  [1014] = {x=-21.274, y=-6.415, z=129.21, rx=179.838, ry=0.326, rz=-127.185, fatherId=FrmDraw[0]}
  [1015] = {x=-21.178, y=-6.199, z=129.218, rx=179.848, ry=0.308, rz=-127.673, fatherId=FrmDraw[0]}
  [1016] = {x=-21.058, y=-5.968, z=129.228, rx=179.861, ry=0.287, rz=-128.317, fatherId=FrmDraw[0]}
  [1017] = {x=-20.945, y=-5.787, z=129.236, rx=179.872, ry=0.268, rz=-128.961, fatherId=FrmDraw[0]}
  [1018] = {x=-20.8, y=-5.61, z=129.247, rx=179.886, ry=0.243, rz=-129.828, fatherId=FrmDraw[0]}
  [1019] = {x=-20.652, y=-5.478, z=129.258, rx=179.9, ry=0.219, rz=-130.741, fatherId=FrmDraw[0]}
  [1020] = {x=-20.476, y=-5.365, z=129.27, rx=179.915, ry=0.19, rz=-131.877, fatherId=FrmDraw[0]}
  [1021] = {x=-20.289, y=-5.287, z=129.282, rx=179.931, ry=0.16, rz=-133.12, fatherId=FrmDraw[0]}
  [1022] = {x=-20.088, y=-5.227, z=129.295, rx=179.946, ry=0.129, rz=-134.508, fatherId=FrmDraw[0]}
  [1023] = {x=-19.895, y=-5.156, z=129.306, rx=179.959, ry=0.102, rz=-135.941, fatherId=FrmDraw[0]}
  [1024] = {x=-19.715, y=-5.077, z=129.317, rx=179.969, ry=0.08, rz=-137.368, fatherId=FrmDraw[0]}
  [1025] = {x=-19.561, y=-4.999, z=129.326, rx=179.976, ry=0.063, rz=-138.682, fatherId=FrmDraw[0]}
  [1026] = {x=-19.427, y=-4.922, z=129.333, rx=179.982, ry=0.05, rz=-139.885, fatherId=FrmDraw[0]}
  [1027] = {x=-19.274, y=-4.826, z=129.341, rx=179.987, ry=0.038, rz=-141.341, fatherId=FrmDraw[0]}
  [1028] = {x=-19.151, y=-4.74, z=129.347, rx=179.99, ry=0.03, rz=-142.591, fatherId=FrmDraw[0]}
  [1029] = {x=-19.043, y=-4.661, z=129.352, rx=179.992, ry=0.024, rz=-143.734, fatherId=FrmDraw[0]}
  [1030] = {x=-18.902, y=-4.55, z=129.359, rx=179.994, ry=0.018, rz=-145.305, fatherId=FrmDraw[0]}
  [1031] = {x=-18.775, y=-4.444, z=129.365, rx=179.996, ry=0.014, rz=-146.807, fatherId=FrmDraw[0]}
  [1032] = {x=-18.658, y=-4.341, z=129.37, rx=179.997, ry=0.011, rz=-148.246, fatherId=FrmDraw[0]}
  [1033] = {x=-18.553, y=-4.238, z=129.374, rx=179.997, ry=0.01, rz=-149.624, fatherId=FrmDraw[0]}
  [1034] = {x=-18.457, y=-4.137, z=129.378, rx=179.997, ry=0.011, rz=-150.951, fatherId=FrmDraw[0]}
  [1035] = {x=-18.37, y=-4.037, z=129.381, rx=179.997, ry=0.012, rz=-152.231, fatherId=FrmDraw[0]}
  [1036] = {x=-18.29, y=-3.938, z=129.384, rx=179.996, ry=0.015, rz=-153.473, fatherId=FrmDraw[0]}
  [1037] = {x=-18.217, y=-3.841, z=129.387, rx=179.996, ry=0.02, rz=-154.679, fatherId=FrmDraw[0]}
  [1038] = {x=-18.151, y=-3.745, z=129.389, rx=179.995, ry=0.025, rz=-155.853, fatherId=FrmDraw[0]}
  [1039] = {x=-18.09, y=-3.651, z=129.39, rx=179.994, ry=0.031, rz=-157, fatherId=FrmDraw[0]}
  [1040] = {x=-18.035, y=-3.558, z=129.392, rx=179.993, ry=0.038, rz=-158.121, fatherId=FrmDraw[0]}
  [1041] = {x=-17.962, y=-3.424, z=129.393, rx=179.991, ry=0.049, rz=-159.732, fatherId=FrmDraw[0]}
  [1042] = {x=-17.898, y=-3.289, z=129.394, rx=179.99, ry=0.063, rz=-161.357, fatherId=FrmDraw[0]}
  [1043] = {x=-17.843, y=-3.162, z=129.394, rx=179.988, ry=0.078, rz=-162.916, fatherId=FrmDraw[0]}
  [1044] = {x=-17.795, y=-3.04, z=129.394, rx=179.987, ry=0.094, rz=-164.461, fatherId=FrmDraw[0]}
  [1045] = {x=-17.752, y=-2.925, z=129.393, rx=179.986, ry=0.111, rz=-165.983, fatherId=FrmDraw[0]}
  [1046] = {x=-17.715, y=-2.816, z=129.392, rx=179.986, ry=0.128, rz=-167.488, fatherId=FrmDraw[0]}
  [1047] = {x=-17.683, y=-2.713, z=129.391, rx=179.986, ry=0.146, rz=-168.981, fatherId=FrmDraw[0]}
  [1048] = {x=-17.654, y=-2.616, z=129.389, rx=179.986, ry=0.164, rz=-170.464, fatherId=FrmDraw[0]}
  [1049] = {x=-17.63, y=-2.525, z=129.388, rx=179.987, ry=0.183, rz=-171.939, fatherId=FrmDraw[0]}
  [1050] = {x=-17.608, y=-2.44, z=129.386, rx=179.988, ry=0.202, rz=-173.407, fatherId=FrmDraw[0]}
  [1051] = {x=-17.59, y=-2.36, z=129.383, rx=179.99, ry=0.221, rz=-174.871, fatherId=FrmDraw[0]}
  [1052] = {x=-17.574, y=-2.286, z=129.381, rx=179.992, ry=0.241, rz=-176.331, fatherId=FrmDraw[0]}
  [1053] = {x=-17.563, y=-2.215, z=129.378, rx=179.995, ry=0.261, rz=-177.777, fatherId=FrmDraw[0]}
  [1054] = {x=-17.557, y=-2.118, z=129.374, rx=179.999, ry=0.29, rz=-179.658, fatherId=FrmDraw[0]}
  [1055] = {x=-17.561, y=-2.02, z=129.368, rx=-179.996, ry=0.321, rz=178.508, fatherId=FrmDraw[0]}
  [1056] = {x=-17.575, y=-1.922, z=129.363, rx=-179.99, ry=0.354, rz=176.715, fatherId=FrmDraw[0]}
  [1057] = {x=-17.597, y=-1.824, z=129.356, rx=-179.983, ry=0.389, rz=174.957, fatherId=FrmDraw[0]}
  [1058] = {x=-17.628, y=-1.725, z=129.349, rx=-179.975, ry=0.426, rz=173.239, fatherId=FrmDraw[0]}
  [1059] = {x=-17.665, y=-1.624, z=129.342, rx=-179.966, ry=0.463, rz=171.562, fatherId=FrmDraw[0]}
  [1060] = {x=-17.705, y=-1.521, z=129.334, rx=-179.956, ry=0.5, rz=169.92, fatherId=FrmDraw[0]}
  [1061] = {x=-17.745, y=-1.417, z=129.327, rx=-179.945, ry=0.534, rz=168.309, fatherId=FrmDraw[0]}
  [1062] = {x=-17.784, y=-1.312, z=129.32, rx=-179.934, ry=0.566, rz=166.727, fatherId=FrmDraw[0]}
  [1063] = {x=-17.822, y=-1.201, z=129.313, rx=-179.923, ry=0.596, rz=165.189, fatherId=FrmDraw[0]}
  [1064] = {x=-17.86, y=-1.084, z=129.307, rx=-179.911, ry=0.624, rz=163.696, fatherId=FrmDraw[0]}
  [1065] = {x=-17.899, y=-0.961, z=129.301, rx=-179.898, ry=0.651, rz=162.246, fatherId=FrmDraw[0]}
  [1066] = {x=-17.941, y=-0.832, z=129.295, rx=-179.886, ry=0.676, rz=160.836, fatherId=FrmDraw[0]}
  [1067] = {x=-17.986, y=-0.698, z=129.289, rx=-179.873, ry=0.702, rz=159.465, fatherId=FrmDraw[0]}
  [1068] = {x=-18.036, y=-0.559, z=129.283, rx=-179.86, ry=0.727, rz=158.13, fatherId=FrmDraw[0]}
  [1069] = {x=-18.09, y=-0.416, z=129.276, rx=-179.846, ry=0.752, rz=156.83, fatherId=FrmDraw[0]}
  [1070] = {x=-18.15, y=-0.268, z=129.269, rx=-179.831, ry=0.779, rz=155.562, fatherId=FrmDraw[0]}
  [1071] = {x=-18.216, y=-0.116, z=129.262, rx=-179.816, ry=0.806, rz=154.324, fatherId=FrmDraw[0]}
  [1072] = {x=-18.289, y=0.038, z=129.255, rx=-179.8, ry=0.835, rz=153.111, fatherId=FrmDraw[0]}
  [1073] = {x=-18.367, y=0.189, z=129.247, rx=-179.784, ry=0.864, rz=151.895, fatherId=FrmDraw[0]}
  [1074] = {x=-18.45, y=0.336, z=129.239, rx=-179.766, ry=0.893, rz=150.671, fatherId=FrmDraw[0]}
  [1075] = {x=-18.536, y=0.479, z=129.231, rx=-179.748, ry=0.922, rz=149.437, fatherId=FrmDraw[0]}
  [1076] = {x=-18.626, y=0.618, z=129.223, rx=-179.729, ry=0.951, rz=148.192, fatherId=FrmDraw[0]}
  [1077] = {x=-18.72, y=0.753, z=129.215, rx=-179.709, ry=0.98, rz=146.934, fatherId=FrmDraw[0]}
  [1078] = {x=-18.817, y=0.883, z=129.206, rx=-179.688, ry=1.008, rz=145.662, fatherId=FrmDraw[0]}
  [1079] = {x=-18.916, y=1.008, z=129.198, rx=-179.667, ry=1.036, rz=144.375, fatherId=FrmDraw[0]}
  [1080] = {x=-19.018, y=1.129, z=129.19, rx=-179.645, ry=1.062, rz=143.071, fatherId=FrmDraw[0]}
  [1081] = {x=-19.123, y=1.245, z=129.182, rx=-179.623, ry=1.088, rz=141.749, fatherId=FrmDraw[0]}
  [1082] = {x=-19.23, y=1.357, z=129.174, rx=-179.599, ry=1.113, rz=140.412, fatherId=FrmDraw[0]}
  [1083] = {x=-19.341, y=1.476, z=129.165, rx=-179.575, ry=1.139, rz=139.111, fatherId=FrmDraw[0]}
  [1084] = {x=-19.398, y=1.539, z=129.161, rx=-179.563, ry=1.152, rz=138.478, fatherId=FrmDraw[0]}
  [1085] = {x=-19.486, y=1.638, z=129.154, rx=-179.545, ry=1.172, rz=137.552, fatherId=FrmDraw[0]}
  [1086] = {x=-19.606, y=1.778, z=129.145, rx=-179.519, ry=1.2, rz=136.36, fatherId=FrmDraw[0]}
  [1087] = {x=-19.729, y=1.929, z=129.136, rx=-179.494, ry=1.229, rz=135.217, fatherId=FrmDraw[0]}
  [1088] = {x=-19.855, y=2.09, z=129.127, rx=-179.468, ry=1.258, rz=134.123, fatherId=FrmDraw[0]}
  [1089] = {x=-19.983, y=2.263, z=129.118, rx=-179.441, ry=1.287, rz=133.079, fatherId=FrmDraw[0]}
  [1090] = {x=-20.112, y=2.448, z=129.108, rx=-179.415, ry=1.316, rz=132.083, fatherId=FrmDraw[0]}
  [1091] = {x=-20.242, y=2.645, z=129.099, rx=-179.389, ry=1.345, rz=131.137, fatherId=FrmDraw[0]}
  [1092] = {x=-20.371, y=2.854, z=129.09, rx=-179.363, ry=1.374, rz=130.24, fatherId=FrmDraw[0]}
  [1093] = {x=-20.499, y=3.072, z=129.082, rx=-179.337, ry=1.401, rz=129.37, fatherId=FrmDraw[0]}
  [1094] = {x=-20.626, y=3.293, z=129.074, rx=-179.313, ry=1.425, rz=128.499, fatherId=FrmDraw[0]}
  [1095] = {x=-20.752, y=3.517, z=129.067, rx=-179.288, ry=1.448, rz=127.626, fatherId=FrmDraw[0]}
  [1096] = {x=-20.879, y=3.742, z=129.06, rx=-179.264, ry=1.468, rz=126.751, fatherId=FrmDraw[0]}
  [1097] = {x=-21.007, y=3.97, z=129.053, rx=-179.24, ry=1.487, rz=125.875, fatherId=FrmDraw[0]}
  [1098] = {x=-21.136, y=4.2, z=129.047, rx=-179.216, ry=1.505, rz=124.995, fatherId=FrmDraw[0]}
  [1099] = {x=-21.268, y=4.431, z=129.041, rx=-179.193, ry=1.522, rz=124.113, fatherId=FrmDraw[0]}
  [1100] = {x=-21.403, y=4.663, z=129.035, rx=-179.169, ry=1.538, rz=123.227, fatherId=FrmDraw[0]}
  [1101] = {x=-21.507, y=4.838, z=129.031, rx=-179.151, ry=1.55, rz=122.561, fatherId=FrmDraw[0]}
  [1102] = {x=-21.643, y=5.061, z=129.025, rx=-179.127, ry=1.566, rz=121.72, fatherId=FrmDraw[0]}
  [1103] = {x=-21.788, y=5.308, z=129.019, rx=-179.102, ry=1.583, rz=120.881, fatherId=FrmDraw[0]}
  [1104] = {x=-21.934, y=5.568, z=129.013, rx=-179.076, ry=1.603, rz=120.103, fatherId=FrmDraw[0]}
  [1105] = {x=-22.076, y=5.838, z=129.007, rx=-179.051, ry=1.623, rz=119.399, fatherId=FrmDraw[0]}
  [1106] = {x=-22.196, y=6.082, z=129.002, rx=-179.03, ry=1.642, rz=118.842, fatherId=FrmDraw[0]}
  [1107] = {x=-22.294, y=6.295, z=128.998, rx=-179.012, ry=1.657, rz=118.41, fatherId=FrmDraw[0]}
  [1108] = {x=-22.427, y=6.609, z=128.993, rx=-178.988, ry=1.679, rz=117.857, fatherId=FrmDraw[0]}
  [1109] = {x=-22.536, y=6.893, z=128.989, rx=-178.968, ry=1.698, rz=117.431, fatherId=FrmDraw[0]}
  [1110] = {x=-22.629, y=7.161, z=128.985, rx=-178.951, ry=1.714, rz=117.087, fatherId=FrmDraw[0]}
  [1111] = {x=-22.717, y=7.442, z=128.983, rx=-178.935, ry=1.73, rz=116.78, fatherId=FrmDraw[0]}
  [1112] = {x=-22.789, y=7.701, z=128.981, rx=-178.922, ry=1.743, rz=116.535, fatherId=FrmDraw[0]}
  [1113] = {x=-22.875, y=8.032, z=128.979, rx=-178.907, ry=1.758, rz=116.241, fatherId=FrmDraw[0]}
  [1114] = {x=-22.941, y=8.301, z=128.978, rx=-178.895, ry=1.768, rz=116.012, fatherId=FrmDraw[0]}
  [1115] = {x=-23.019, y=8.644, z=128.977, rx=-178.882, ry=1.78, rz=115.735, fatherId=FrmDraw[0]}
  [1116] = {x=-23.079, y=8.922, z=128.976, rx=-178.873, ry=1.787, rz=115.52, fatherId=FrmDraw[0]}
  [1117] = {x=-23.152, y=9.275, z=128.976, rx=-178.861, ry=1.796, rz=115.261, fatherId=FrmDraw[0]}
  [1118] = {x=-23.214, y=9.597, z=128.977, rx=-178.852, ry=1.803, rz=115.036, fatherId=FrmDraw[0]}
  [1119] = {x=-23.276, y=9.924, z=128.977, rx=-178.843, ry=1.81, rz=114.819, fatherId=FrmDraw[0]}
  [1120] = {x=-23.329, y=10.217, z=128.978, rx=-178.835, ry=1.815, rz=114.634, fatherId=FrmDraw[0]}
  [1121] = {x=-23.395, y=10.588, z=128.979, rx=-178.826, ry=1.822, rz=114.411, fatherId=FrmDraw[0]}
  [1122] = {x=-23.446, y=10.887, z=128.98, rx=-178.819, ry=1.827, rz=114.24, fatherId=FrmDraw[0]}
  [1123] = {x=-23.512, y=11.264, z=128.981, rx=-178.81, ry=1.834, rz=114.035, fatherId=FrmDraw[0]}
  [1124] = {x=-23.565, y=11.566, z=128.982, rx=-178.802, ry=1.84, rz=113.87, fatherId=FrmDraw[0]}
  [1125] = {x=-23.634, y=11.944, z=128.983, rx=-178.792, ry=1.847, rz=113.662, fatherId=FrmDraw[0]}
  [1126] = {x=-23.698, y=12.284, z=128.984, rx=-178.784, ry=1.854, rz=113.474, fatherId=FrmDraw[0]}
  [1127] = {x=-23.763, y=12.625, z=128.985, rx=-178.775, ry=1.861, rz=113.284, fatherId=FrmDraw[0]}
  [1128] = {x=-23.822, y=12.928, z=128.986, rx=-178.767, ry=1.866, rz=113.114, fatherId=FrmDraw[0]}
  [1129] = {x=-23.897, y=13.307, z=128.988, rx=-178.757, ry=1.874, rz=112.9, fatherId=FrmDraw[0]}
  [1130] = {x=-23.959, y=13.611, z=128.989, rx=-178.75, ry=1.879, rz=112.728, fatherId=FrmDraw[0]}
  [1131] = {x=-24.038, y=13.992, z=128.99, rx=-178.74, ry=1.886, rz=112.511, fatherId=FrmDraw[0]}
  [1132] = {x=-24.102, y=14.297, z=128.992, rx=-178.732, ry=1.892, rz=112.336, fatherId=FrmDraw[0]}
  [1133] = {x=-24.183, y=14.679, z=128.994, rx=-178.722, ry=1.898, rz=112.116, fatherId=FrmDraw[0]}
  [1134] = {x=-24.257, y=15.023, z=128.995, rx=-178.714, ry=1.904, rz=111.916, fatherId=FrmDraw[0]}
  [1135] = {x=-24.333, y=15.369, z=128.997, rx=-178.705, ry=1.909, rz=111.714, fatherId=FrmDraw[0]}
  [1136] = {x=-24.401, y=15.677, z=128.999, rx=-178.698, ry=1.913, rz=111.534, fatherId=FrmDraw[0]}
  [1137] = {x=-24.487, y=16.063, z=129.001, rx=-178.689, ry=1.919, rz=111.306, fatherId=FrmDraw[0]}
  [1138] = {x=-24.556, y=16.372, z=129.002, rx=-178.682, ry=1.922, rz=111.123, fatherId=FrmDraw[0]}
  [1139] = {x=-24.644, y=16.761, z=129.005, rx=-178.673, ry=1.926, rz=110.892, fatherId=FrmDraw[0]}
  [1140] = {x=-24.715, y=17.073, z=129.007, rx=-178.667, ry=1.929, rz=110.705, fatherId=FrmDraw[0]}
  [1141] = {x=-24.805, y=17.464, z=129.009, rx=-178.659, ry=1.932, rz=110.47, fatherId=FrmDraw[0]}
  [1142] = {x=-24.887, y=17.817, z=129.012, rx=-178.652, ry=1.934, rz=110.257, fatherId=FrmDraw[0]}
  [1143] = {x=-24.969, y=18.172, z=129.014, rx=-178.646, ry=1.936, rz=110.042, fatherId=FrmDraw[0]}
  [1144] = {x=-25.042, y=18.489, z=129.017, rx=-178.64, ry=1.936, rz=109.85, fatherId=FrmDraw[0]}
  [1145] = {x=-25.134, y=18.887, z=129.02, rx=-178.634, ry=1.937, rz=109.61, fatherId=FrmDraw[0]}
  [1146] = {x=-25.207, y=19.207, z=129.022, rx=-178.629, ry=1.937, rz=109.419, fatherId=FrmDraw[0]}
  [1147] = {x=-25.3, y=19.609, z=129.025, rx=-178.623, ry=1.936, rz=109.18, fatherId=FrmDraw[0]}
  [1148] = {x=-25.376, y=19.932, z=129.028, rx=-178.619, ry=1.936, rz=108.99, fatherId=FrmDraw[0]}
  [1149] = {x=-25.472, y=20.336, z=129.031, rx=-178.613, ry=1.936, rz=108.752, fatherId=FrmDraw[0]}
  [1150] = {x=-25.562, y=20.701, z=129.034, rx=-178.607, ry=1.937, rz=108.54, fatherId=FrmDraw[0]}
  [1151] = {x=-25.653, y=21.066, z=129.037, rx=-178.6, ry=1.938, rz=108.327, fatherId=FrmDraw[0]}
  [1152] = {x=-25.737, y=21.39, z=129.039, rx=-178.594, ry=1.94, rz=108.139, fatherId=FrmDraw[0]}
  [1153] = {x=-25.846, y=21.795, z=129.042, rx=-178.586, ry=1.943, rz=107.904, fatherId=FrmDraw[0]}
  [1154] = {x=-25.936, y=22.119, z=129.045, rx=-178.578, ry=1.947, rz=107.719, fatherId=FrmDraw[0]}
  [1155] = {x=-26.047, y=22.528, z=129.048, rx=-178.568, ry=1.953, rz=107.502, fatherId=FrmDraw[0]}
  [1156] = {x=-26.133, y=22.859, z=129.051, rx=-178.559, ry=1.959, rz=107.339, fatherId=FrmDraw[0]}
  [1157] = {x=-26.233, y=23.28, z=129.054, rx=-178.55, ry=1.965, rz=107.151, fatherId=FrmDraw[0]}
  [1158] = {x=-26.315, y=23.667, z=129.058, rx=-178.543, ry=1.969, rz=106.995, fatherId=FrmDraw[0]}
  [1159] = {x=-26.388, y=24.063, z=129.062, rx=-178.537, ry=1.972, rz=106.853, fatherId=FrmDraw[0]}
  [1160] = {x=-26.452, y=24.5, z=129.067, rx=-178.534, ry=1.971, rz=106.716, fatherId=FrmDraw[0]}
  [1161] = {x=-26.494, y=24.888, z=129.071, rx=-178.534, ry=1.967, rz=106.61, fatherId=FrmDraw[0]}
  [1162] = {x=-26.526, y=25.353, z=129.077, rx=-178.539, ry=1.957, rz=106.502, fatherId=FrmDraw[0]}
  [1163] = {x=-26.572, y=25.741, z=129.081, rx=-178.546, ry=1.942, rz=106.344, fatherId=FrmDraw[0]}
  [1164] = {x=-26.564, y=25.744, z=129.498, rx=-178.546, ry=1.941, rz=106.357, fatherId=FrmDraw[0]}
  [1165] = {x=-26.557, y=25.747, z=129.915, rx=-178.547, ry=1.941, rz=106.37, fatherId=FrmDraw[0]}
  [1166] = {x=-26.549, y=25.75, z=130.379, rx=-178.548, ry=1.941, rz=106.384, fatherId=FrmDraw[0]}
  [1167] = {x=-26.544, y=25.753, z=130.721, rx=-178.548, ry=1.941, rz=106.395, fatherId=FrmDraw[0]}
  [1168] = {x=-26.538, y=25.755, z=131.062, rx=-178.548, ry=1.94, rz=106.405, fatherId=FrmDraw[0]}
  [1169] = {x=-26.53, y=25.758, z=131.484, rx=-178.549, ry=1.94, rz=106.418, fatherId=FrmDraw[0]}
  [1170] = {x=-26.522, y=25.761, z=131.958, rx=-178.55, ry=1.94, rz=106.433, fatherId=FrmDraw[0]}
  [1171] = {x=-26.515, y=25.765, z=132.407, rx=-178.55, ry=1.94, rz=106.447, fatherId=FrmDraw[0]}
  [1172] = {x=-26.508, y=25.767, z=132.773, rx=-178.551, ry=1.939, rz=106.458, fatherId=FrmDraw[0]}
  [1173] = {x=-26.502, y=25.77, z=133.139, rx=-178.551, ry=1.939, rz=106.47, fatherId=FrmDraw[0]}
  [1174] = {x=-26.473, y=25.37, z=133.135, rx=-178.543, ry=1.955, rz=106.597, fatherId=FrmDraw[0]}
  [1175] = {x=-26.468, y=24.887, z=133.129, rx=-178.537, ry=1.964, rz=106.651, fatherId=FrmDraw[0]}
  [1176] = {x=-26.444, y=24.487, z=133.124, rx=-178.536, ry=1.968, rz=106.718, fatherId=FrmDraw[0]}
  [1177] = {x=-26.396, y=24.038, z=133.119, rx=-178.539, ry=1.968, rz=106.819, fatherId=FrmDraw[0]}
  [1178] = {x=-26.339, y=23.664, z=133.114, rx=-178.544, ry=1.965, rz=106.926, fatherId=FrmDraw[0]}
  [1179] = {x=-26.258, y=23.242, z=133.11, rx=-178.552, ry=1.96, rz=107.072, fatherId=FrmDraw[0]}
  [1180] = {x=-26.16, y=22.819, z=133.107, rx=-178.561, ry=1.953, rz=107.25, fatherId=FrmDraw[0]}
  [1181] = {x=-26.074, y=22.488, z=133.104, rx=-178.57, ry=1.947, rz=107.41, fatherId=FrmDraw[0]}
  [1182] = {x=-25.959, y=22.082, z=133.101, rx=-178.58, ry=1.941, rz=107.634, fatherId=FrmDraw[0]}
  [1183] = {x=-25.864, y=21.762, z=133.099, rx=-178.588, ry=1.937, rz=107.83, fatherId=FrmDraw[0]}
  [1184] = {x=-25.749, y=21.362, z=133.096, rx=-178.597, ry=1.933, rz=108.077, fatherId=FrmDraw[0]}
  [1185] = {x=-25.662, y=21.04, z=133.093, rx=-178.603, ry=1.932, rz=108.273, fatherId=FrmDraw[0]}
  [1186] = {x=-25.557, y=20.637, z=133.09, rx=-178.61, ry=1.931, rz=108.517, fatherId=FrmDraw[0]}
  [1187] = {x=-25.476, y=20.315, z=133.088, rx=-178.616, ry=1.93, rz=108.711, fatherId=FrmDraw[0]}
  [1188] = {x=-25.379, y=19.911, z=133.085, rx=-178.622, ry=1.931, rz=108.952, fatherId=FrmDraw[0]}
  [1189] = {x=-25.303, y=19.589, z=133.082, rx=-178.626, ry=1.931, rz=109.143, fatherId=FrmDraw[0]}
  [1190] = {x=-25.21, y=19.187, z=133.079, rx=-178.632, ry=1.931, rz=109.381, fatherId=FrmDraw[0]}
  [1191] = {x=-25.137, y=18.866, z=133.076, rx=-178.637, ry=1.931, rz=109.57, fatherId=FrmDraw[0]}
  [1192] = {x=-25.047, y=18.466, z=133.073, rx=-178.643, ry=1.931, rz=109.805, fatherId=FrmDraw[0]}
  [1193] = {x=-24.975, y=18.148, z=133.071, rx=-178.648, ry=1.93, rz=109.992, fatherId=FrmDraw[0]}
  [1194] = {x=-24.886, y=17.752, z=133.068, rx=-178.655, ry=1.929, rz=110.224, fatherId=FrmDraw[0]}
  [1195] = {x=-24.815, y=17.437, z=133.066, rx=-178.661, ry=1.927, rz=110.408, fatherId=FrmDraw[0]}
  [1196] = {x=-24.727, y=17.044, z=133.063, rx=-178.669, ry=1.924, rz=110.637, fatherId=FrmDraw[0]}
  [1197] = {x=-24.656, y=16.732, z=133.061, rx=-178.676, ry=1.921, rz=110.819, fatherId=FrmDraw[0]}
  [1198] = {x=-24.569, y=16.342, z=133.059, rx=-178.684, ry=1.916, rz=111.045, fatherId=FrmDraw[0]}
  [1199] = {x=-24.499, y=16.032, z=133.057, rx=-178.691, ry=1.912, rz=111.225, fatherId=FrmDraw[0]}
  [1200] = {x=-24.414, y=15.645, z=133.055, rx=-178.7, ry=1.907, rz=111.449, fatherId=FrmDraw[0]}
  [1201] = {x=-24.346, y=15.337, z=133.053, rx=-178.708, ry=1.902, rz=111.626, fatherId=FrmDraw[0]}
  [1202] = {x=-24.262, y=14.953, z=133.052, rx=-178.717, ry=1.896, rz=111.847, fatherId=FrmDraw[0]}
  [1203] = {x=-24.196, y=14.646, z=133.05, rx=-178.725, ry=1.891, rz=112.023, fatherId=FrmDraw[0]}
  [1204] = {x=-24.114, y=14.264, z=133.048, rx=-178.734, ry=1.885, rz=112.241, fatherId=FrmDraw[0]}
  [1205] = {x=-24.05, y=13.959, z=133.047, rx=-178.742, ry=1.879, rz=112.414, fatherId=FrmDraw[0]}
  [1206] = {x=-23.971, y=13.578, z=133.046, rx=-178.752, ry=1.872, rz=112.63, fatherId=FrmDraw[0]}
  [1207] = {x=-23.909, y=13.274, z=133.044, rx=-178.76, ry=1.866, rz=112.801, fatherId=FrmDraw[0]}
  [1208] = {x=-23.833, y=12.895, z=133.043, rx=-178.77, ry=1.859, rz=113.015, fatherId=FrmDraw[0]}
  [1209] = {x=-23.773, y=12.592, z=133.042, rx=-178.778, ry=1.853, rz=113.184, fatherId=FrmDraw[0]}
  [1210] = {x=-23.7, y=12.214, z=133.041, rx=-178.787, ry=1.846, rz=113.395, fatherId=FrmDraw[0]}
  [1211] = {x=-23.643, y=11.912, z=133.04, rx=-178.795, ry=1.84, rz=113.563, fatherId=FrmDraw[0]}
  [1212] = {x=-23.574, y=11.535, z=133.038, rx=-178.804, ry=1.833, rz=113.772, fatherId=FrmDraw[0]}
  [1213] = {x=-23.52, y=11.233, z=133.038, rx=-178.812, ry=1.827, rz=113.938, fatherId=FrmDraw[0]}
  [1214] = {x=-23.454, y=10.857, z=133.036, rx=-178.821, ry=1.821, rz=114.145, fatherId=FrmDraw[0]}
  [1215] = {x=-23.401, y=10.558, z=133.036, rx=-178.828, ry=1.815, rz=114.316, fatherId=FrmDraw[0]}
  [1216] = {x=-23.336, y=10.187, z=133.035, rx=-178.837, ry=1.809, rz=114.537, fatherId=FrmDraw[0]}
  [1217] = {x=-23.283, y=9.892, z=133.034, rx=-178.845, ry=1.803, rz=114.719, fatherId=FrmDraw[0]}
  [1218] = {x=-23.216, y=9.528, z=133.033, rx=-178.855, ry=1.796, rz=114.953, fatherId=FrmDraw[0]}
  [1219] = {x=-23.161, y=9.24, z=133.033, rx=-178.863, ry=1.79, rz=115.146, fatherId=FrmDraw[0]}
  [1220] = {x=-23.09, y=8.884, z=133.033, rx=-178.874, ry=1.781, rz=115.394, fatherId=FrmDraw[0]}
  [1221] = {x=-23.031, y=8.602, z=133.033, rx=-178.883, ry=1.773, rz=115.597, fatherId=FrmDraw[0]}
  [1222] = {x=-22.955, y=8.255, z=133.034, rx=-178.896, ry=1.762, rz=115.857, fatherId=FrmDraw[0]}
  [1223] = {x=-22.891, y=7.982, z=133.035, rx=-178.907, ry=1.751, rz=116.07, fatherId=FrmDraw[0]}
  [1224] = {x=-22.807, y=7.645, z=133.037, rx=-178.922, ry=1.736, rz=116.343, fatherId=FrmDraw[0]}
  [1225] = {x=-22.736, y=7.382, z=133.039, rx=-178.935, ry=1.723, rz=116.573, fatherId=FrmDraw[0]}
  [1226] = {x=-22.64, y=7.067, z=133.042, rx=-178.953, ry=1.706, rz=116.902, fatherId=FrmDraw[0]}
  [1227] = {x=-22.558, y=6.827, z=133.044, rx=-178.968, ry=1.691, rz=117.201, fatherId=FrmDraw[0]}
  [1228] = {x=-22.462, y=6.568, z=133.048, rx=-178.985, ry=1.675, rz=117.574, fatherId=FrmDraw[0]}
  [1229] = {x=-22.361, y=6.321, z=133.052, rx=-179.003, ry=1.659, rz=117.987, fatherId=FrmDraw[0]}
  [1230] = {x=-22.245, y=6.06, z=133.056, rx=-179.024, ry=1.641, rz=118.489, fatherId=FrmDraw[0]}
  [1231] = {x=-22.106, y=5.772, z=133.062, rx=-179.048, ry=1.621, rz=119.134, fatherId=FrmDraw[0]}
  [1232] = {x=-22.005, y=5.577, z=133.066, rx=-179.065, ry=1.607, rz=119.631, fatherId=FrmDraw[0]}
  [1233] = {x=-21.884, y=5.355, z=133.071, rx=-179.087, ry=1.591, rz=120.269, fatherId=FrmDraw[0]}
  [1234] = {x=-21.741, y=5.109, z=133.077, rx=-179.111, ry=1.573, rz=121.067, fatherId=FrmDraw[0]}
  [1235] = {x=-21.604, y=4.885, z=133.082, rx=-179.135, ry=1.558, rz=121.894, fatherId=FrmDraw[0]}
  [1236] = {x=-21.497, y=4.71, z=133.087, rx=-179.153, ry=1.546, rz=122.563, fatherId=FrmDraw[0]}
  [1237] = {x=-21.358, y=4.477, z=133.093, rx=-179.177, ry=1.529, rz=123.448, fatherId=FrmDraw[0]}
  [1238] = {x=-21.222, y=4.246, z=133.099, rx=-179.201, ry=1.512, rz=124.328, fatherId=FrmDraw[0]}
  [1239] = {x=-21.089, y=4.015, z=133.105, rx=-179.226, ry=1.494, rz=125.202, fatherId=FrmDraw[0]}
  [1240] = {x=-20.958, y=3.785, z=133.112, rx=-179.25, ry=1.474, rz=126.07, fatherId=FrmDraw[0]}
  [1241] = {x=-20.827, y=3.558, z=133.119, rx=-179.274, ry=1.453, rz=126.934, fatherId=FrmDraw[0]}
  [1242] = {x=-20.698, y=3.331, z=133.127, rx=-179.299, ry=1.43, rz=127.794, fatherId=FrmDraw[0]}
  [1243] = {x=-20.568, y=3.107, z=133.134, rx=-179.324, ry=1.405, rz=128.65, fatherId=FrmDraw[0]}
  [1244] = {x=-20.438, y=2.885, z=133.143, rx=-179.35, ry=1.378, rz=129.501, fatherId=FrmDraw[0]}
  [1245] = {x=-20.307, y=2.668, z=133.151, rx=-179.376, ry=1.35, rz=130.368, fatherId=FrmDraw[0]}
  [1246] = {x=-20.176, y=2.465, z=133.16, rx=-179.402, ry=1.321, rz=131.285, fatherId=FrmDraw[0]}
  [1247] = {x=-20.046, y=2.274, z=133.17, rx=-179.428, ry=1.292, rz=132.254, fatherId=FrmDraw[0]}
  [1248] = {x=-19.917, y=2.095, z=133.179, rx=-179.454, ry=1.263, rz=133.274, fatherId=FrmDraw[0]}
  [1249] = {x=-19.79, y=1.928, z=133.188, rx=-179.48, ry=1.235, rz=134.346, fatherId=FrmDraw[0]}
  [1250] = {x=-19.665, y=1.773, z=133.197, rx=-179.506, ry=1.207, rz=135.469, fatherId=FrmDraw[0]}
  [1251] = {x=-19.544, y=1.629, z=133.206, rx=-179.531, ry=1.179, rz=136.643, fatherId=FrmDraw[0]}
  [1252] = {x=-19.426, y=1.495, z=133.215, rx=-179.556, ry=1.152, rz=137.868, fatherId=FrmDraw[0]}
  [1253] = {x=-19.311, y=1.372, z=133.223, rx=-179.58, ry=1.126, rz=139.143, fatherId=FrmDraw[0]}
  [1254] = {x=-19.201, y=1.258, z=133.232, rx=-179.604, ry=1.101, rz=140.467, fatherId=FrmDraw[0]}
  [1255] = {x=-19.092, y=1.145, z=133.24, rx=-179.627, ry=1.076, rz=141.797, fatherId=FrmDraw[0]}
  [1256] = {x=-18.986, y=1.027, z=133.248, rx=-179.65, ry=1.049, rz=143.108, fatherId=FrmDraw[0]}
  [1257] = {x=-18.881, y=0.905, z=133.257, rx=-179.672, ry=1.021, rz=144.403, fatherId=FrmDraw[0]}
  [1258] = {x=-18.779, y=0.779, z=133.265, rx=-179.694, ry=0.992, rz=145.683, fatherId=FrmDraw[0]}
  [1259] = {x=-18.679, y=0.649, z=133.274, rx=-179.714, ry=0.962, rz=146.949, fatherId=FrmDraw[0]}
  [1260] = {x=-18.583, y=0.514, z=133.282, rx=-179.734, ry=0.933, rz=148.203, fatherId=FrmDraw[0]}
  [1261] = {x=-18.49, y=0.376, z=133.291, rx=-179.754, ry=0.902, rz=149.446, fatherId=FrmDraw[0]}
  [1262] = {x=-18.401, y=0.233, z=133.299, rx=-179.772, ry=0.872, rz=150.68, fatherId=FrmDraw[0]}
  [1263] = {x=-18.317, y=0.087, z=133.307, rx=-179.789, ry=0.842, rz=151.906, fatherId=FrmDraw[0]}
  [1264] = {x=-18.238, y=-0.063, z=133.315, rx=-179.806, ry=0.813, rz=153.125, fatherId=FrmDraw[0]}
  [1265] = {x=-18.165, y=-0.214, z=133.322, rx=-179.822, ry=0.784, rz=154.356, fatherId=FrmDraw[0]}
  [1266] = {x=-18.1, y=-0.361, z=133.329, rx=-179.836, ry=0.757, rz=155.614, fatherId=FrmDraw[0]}
  [1267] = {x=-18.04, y=-0.506, z=133.336, rx=-179.851, ry=0.731, rz=156.898, fatherId=FrmDraw[0]}
  [1268] = {x=-17.986, y=-0.647, z=133.343, rx=-179.864, ry=0.705, rz=158.212, fatherId=FrmDraw[0]}
  [1269] = {x=-17.937, y=-0.784, z=133.349, rx=-179.877, ry=0.68, rz=159.558, fatherId=FrmDraw[0]}
  [1270] = {x=-17.891, y=-0.916, z=133.355, rx=-179.89, ry=0.654, rz=160.936, fatherId=FrmDraw[0]}
  [1271] = {x=-17.847, y=-1.044, z=133.361, rx=-179.903, ry=0.627, rz=162.349, fatherId=FrmDraw[0]}
  [1272] = {x=-17.806, y=-1.167, z=133.368, rx=-179.915, ry=0.6, rz=163.8, fatherId=FrmDraw[0]}
  [1273] = {x=-17.765, y=-1.285, z=133.374, rx=-179.926, ry=0.571, rz=165.289, fatherId=FrmDraw[0]}
  [1274] = {x=-17.724, y=-1.398, z=133.381, rx=-179.938, ry=0.539, rz=166.819, fatherId=FrmDraw[0]}
  [1275] = {x=-17.681, y=-1.507, z=133.388, rx=-179.949, ry=0.506, rz=168.386, fatherId=FrmDraw[0]}
  [1276] = {x=-17.639, y=-1.613, z=133.396, rx=-179.959, ry=0.47, rz=169.99, fatherId=FrmDraw[0]}
  [1277] = {x=-17.6, y=-1.716, z=133.403, rx=-179.968, ry=0.434, rz=171.637, fatherId=FrmDraw[0]}
  [1278] = {x=-17.567, y=-1.814, z=133.41, rx=-179.977, ry=0.398, rz=173.33, fatherId=FrmDraw[0]}
  [1279] = {x=-17.542, y=-1.909, z=133.417, rx=-179.984, ry=0.364, rz=175.074, fatherId=FrmDraw[0]}
  [1280] = {x=-17.526, y=-2.004, z=133.423, rx=-179.991, ry=0.331, rz=176.854, fatherId=FrmDraw[0]}
  [1281] = {x=-17.519, y=-2.098, z=133.428, rx=-179.997, ry=0.3, rz=178.672, fatherId=FrmDraw[0]}
  [1282] = {x=-17.521, y=-2.191, z=133.433, rx=179.999, ry=0.271, rz=-179.467, fatherId=FrmDraw[0]}
  [1283] = {x=-17.533, y=-2.282, z=133.436, rx=179.995, ry=0.244, rz=-177.556, fatherId=FrmDraw[0]}
  [1284] = {x=-17.547, y=-2.352, z=133.439, rx=179.992, ry=0.225, rz=-176.097, fatherId=FrmDraw[0]}
  [1285] = {x=-17.564, y=-2.427, z=133.441, rx=179.99, ry=0.206, rz=-174.634, fatherId=FrmDraw[0]}
  [1286] = {x=-17.584, y=-2.507, z=133.444, rx=179.989, ry=0.187, rz=-173.168, fatherId=FrmDraw[0]}
  [1287] = {x=-17.606, y=-2.592, z=133.446, rx=179.988, ry=0.168, rz=-171.696, fatherId=FrmDraw[0]}
  [1288] = {x=-17.632, y=-2.683, z=133.447, rx=179.987, ry=0.149, rz=-170.217, fatherId=FrmDraw[0]}
  [1289] = {x=-17.662, y=-2.781, z=133.449, rx=179.987, ry=0.131, rz=-168.728, fatherId=FrmDraw[0]}
  [1290] = {x=-17.695, y=-2.884, z=133.45, rx=179.987, ry=0.114, rz=-167.229, fatherId=FrmDraw[0]}
  [1291] = {x=-17.734, y=-2.992, z=133.451, rx=179.988, ry=0.096, rz=-165.715, fatherId=FrmDraw[0]}
  [1292] = {x=-17.778, y=-3.107, z=133.451, rx=179.989, ry=0.08, rz=-164.183, fatherId=FrmDraw[0]}
  [1293] = {x=-17.828, y=-3.228, z=133.452, rx=179.99, ry=0.065, rz=-162.63, fatherId=FrmDraw[0]}
  [1294] = {x=-17.885, y=-3.352, z=133.451, rx=179.992, ry=0.05, rz=-161.071, fatherId=FrmDraw[0]}
  [1295] = {x=-17.941, y=-3.46, z=133.45, rx=179.993, ry=0.039, rz=-159.719, fatherId=FrmDraw[0]}
  [1296] = {x=-18.004, y=-3.572, z=133.449, rx=179.994, ry=0.03, rz=-158.326, fatherId=FrmDraw[0]}
  [1297] = {x=-18.086, y=-3.702, z=133.447, rx=179.996, ry=0.02, rz=-156.692, fatherId=FrmDraw[0]}
  [1298] = {x=-18.149, y=-3.793, z=133.445, rx=179.997, ry=0.015, rz=-155.54, fatherId=FrmDraw[0]}
  [1299] = {x=-18.239, y=-3.912, z=133.442, rx=179.998, ry=0.009, rz=-154.009, fatherId=FrmDraw[0]}
  [1300] = {x=-18.34, y=-4.035, z=133.439, rx=179.999, ry=0.005, rz=-152.408, fatherId=FrmDraw[0]}
  [1301] = {x=-18.428, y=-4.132, z=133.435, rx=179.999, ry=0.003, rz=-151.121, fatherId=FrmDraw[0]}
  [1302] = {x=-18.524, y=-4.23, z=133.432, rx=179.999, ry=0.003, rz=-149.79, fatherId=FrmDraw[0]}
  [1303] = {x=-18.629, y=-4.329, z=133.427, rx=179.999, ry=0.003, rz=-148.406, fatherId=FrmDraw[0]}
  [1304] = {x=-18.745, y=-4.429, z=133.422, rx=179.998, ry=0.006, rz=-146.962, fatherId=FrmDraw[0]}
  [1305] = {x=-18.872, y=-4.532, z=133.417, rx=179.997, ry=0.01, rz=-145.455, fatherId=FrmDraw[0]}
  [1306] = {x=-19.013, y=-4.638, z=133.41, rx=179.995, ry=0.016, rz=-143.875, fatherId=FrmDraw[0]}
  [1307] = {x=-19.139, y=-4.724, z=133.404, rx=179.992, ry=0.023, rz=-142.545, fatherId=FrmDraw[0]}
  [1308] = {x=-19.271, y=-4.808, z=133.397, rx=179.989, ry=0.032, rz=-141.215, fatherId=FrmDraw[0]}
  [1309] = {x=-19.406, y=-4.884, z=133.39, rx=179.984, ry=0.043, rz=-139.934, fatherId=FrmDraw[0]}
  [1310] = {x=-19.568, y=-4.965, z=133.382, rx=179.978, ry=0.059, rz=-138.494, fatherId=FrmDraw[0]}
  [1311] = {x=-19.744, y=-5.039, z=133.372, rx=179.969, ry=0.079, rz=-137.025, fatherId=FrmDraw[0]}
  [1312] = {x=-19.888, y=-5.091, z=133.364, rx=179.961, ry=0.097, rz=-135.888, fatherId=FrmDraw[0]}
  [1313] = {x=-20.084, y=-5.149, z=133.352, rx=179.948, ry=0.124, rz=-134.438, fatherId=FrmDraw[0]}
  [1314] = {x=-20.26, y=-5.193, z=133.341, rx=179.935, ry=0.151, rz=-133.204, fatherId=FrmDraw[0]}
  [1315] = {x=-20.439, y=-5.265, z=133.33, rx=179.921, ry=0.178, rz=-131.98, fatherId=FrmDraw[0]}
  [1316] = {x=-20.607, y=-5.369, z=133.318, rx=179.907, ry=0.204, rz=-130.856, fatherId=FrmDraw[0]}
  [1317] = {x=-20.778, y=-5.525, z=133.306, rx=179.892, ry=0.231, rz=-129.751, fatherId=FrmDraw[0]}
  [1318] = {x=-20.919, y=-5.704, z=133.296, rx=179.879, ry=0.253, rz=-128.881, fatherId=FrmDraw[0]}
  [1319] = {x=-21.06, y=-5.945, z=133.285, rx=179.866, ry=0.275, rz=-128.052, fatherId=FrmDraw[0]}
  [1320] = {x=-21.152, y=-6.136, z=133.277, rx=179.857, ry=0.291, rz=-127.539, fatherId=FrmDraw[0]}
  [1321] = {x=-21.259, y=-6.406, z=133.268, rx=179.846, ry=0.308, rz=-126.971, fatherId=FrmDraw[0]}
  [1322] = {x=-21.345, y=-6.69, z=133.26, rx=179.838, ry=0.322, rz=-126.521, fatherId=FrmDraw[0]}
  [1323] = {x=-21.423, y=-7.06, z=133.252, rx=179.831, ry=0.333, rz=-126.105, fatherId=FrmDraw[0]}
  [1324] = {x=-21.466, y=-7.358, z=133.247, rx=179.828, ry=0.337, rz=-125.86, fatherId=FrmDraw[0]}
  [1325] = {x=-21.508, y=-7.649, z=133.243, rx=179.825, ry=0.341, rz=-125.618, fatherId=FrmDraw[0]}
  [1326] = {x=-21.565, y=-8.012, z=133.237, rx=179.821, ry=0.346, rz=-125.296, fatherId=FrmDraw[0]}
  [1327] = {x=-21.629, y=-8.388, z=133.231, rx=179.818, ry=0.35, rz=-124.942, fatherId=FrmDraw[0]}
  [1328] = {x=-21.681, y=-8.672, z=133.226, rx=179.815, ry=0.354, rz=-124.658, fatherId=FrmDraw[0]}
  [1329] = {x=-21.752, y=-9.03, z=133.22, rx=179.811, ry=0.358, rz=-124.281, fatherId=FrmDraw[0]}
  [1330] = {x=-21.827, y=-9.376, z=133.214, rx=179.807, ry=0.362, rz=-123.894, fatherId=FrmDraw[0]}
  [1331] = {x=-21.815, y=-9.377, z=133.632, rx=179.81, ry=0.357, rz=-123.893, fatherId=FrmDraw[0]}
  [1332] = {x=-21.804, y=-9.377, z=134.05, rx=179.813, ry=0.352, rz=-123.892, fatherId=FrmDraw[0]}
  [1333] = {x=-21.791, y=-9.378, z=134.514, rx=179.816, ry=0.346, rz=-123.891, fatherId=FrmDraw[0]}
  [1334] = {x=-21.781, y=-9.378, z=134.858, rx=179.818, ry=0.342, rz=-123.89, fatherId=FrmDraw[0]}
  [1335] = {x=-21.771, y=-9.379, z=135.201, rx=179.82, ry=0.337, rz=-123.889, fatherId=FrmDraw[0]}
  [1336] = {x=-21.759, y=-9.379, z=135.622, rx=179.823, ry=0.332, rz=-123.888, fatherId=FrmDraw[0]}
  [1337] = {x=-21.745, y=-9.38, z=136.11, rx=179.826, ry=0.326, rz=-123.887, fatherId=FrmDraw[0]}
  [1338] = {x=-21.731, y=-9.381, z=136.566, rx=179.829, ry=0.321, rz=-123.886, fatherId=FrmDraw[0]}
  [1339] = {x=-21.72, y=-9.382, z=136.955, rx=179.832, ry=0.316, rz=-123.885, fatherId=FrmDraw[0]}
  [1340] = {x=-21.708, y=-9.383, z=137.344, rx=179.834, ry=0.311, rz=-123.885, fatherId=FrmDraw[0]}
  [1341] = {x=-21.638, y=-9.082, z=137.35, rx=179.838, ry=0.306, rz=-124.224, fatherId=FrmDraw[0]}
  [1342] = {x=-21.559, y=-8.708, z=137.357, rx=179.843, ry=0.299, rz=-124.623, fatherId=FrmDraw[0]}
  [1343] = {x=-21.487, y=-8.334, z=137.364, rx=179.847, ry=0.294, rz=-124.996, fatherId=FrmDraw[0]}
  [1344] = {x=-21.426, y=-7.977, z=137.37, rx=179.851, ry=0.289, rz=-125.331, fatherId=FrmDraw[0]}
  [1345] = {x=-21.369, y=-7.595, z=137.376, rx=179.854, ry=0.285, rz=-125.665, fatherId=FrmDraw[0]}
  [1346] = {x=-21.327, y=-7.281, z=137.381, rx=179.856, ry=0.282, rz=-125.924, fatherId=FrmDraw[0]}
  [1347] = {x=-21.29, y=-6.974, z=137.386, rx=179.858, ry=0.28, rz=-126.165, fatherId=FrmDraw[0]}
  [1348] = {x=-21.231, y=-6.634, z=137.392, rx=179.862, ry=0.274, rz=-126.52, fatherId=FrmDraw[0]}
  [1349] = {x=-21.143, y=-6.303, z=137.4, rx=179.869, ry=0.262, rz=-127.029, fatherId=FrmDraw[0]}
  [1350] = {x=-21.063, y=-6.078, z=137.407, rx=179.876, ry=0.251, rz=-127.5, fatherId=FrmDraw[0]}
  [1351] = {x=-20.956, y=-5.841, z=137.416, rx=179.886, ry=0.235, rz=-128.144, fatherId=FrmDraw[0]}
  [1352] = {x=-20.846, y=-5.646, z=137.424, rx=179.895, ry=0.22, rz=-128.839, fatherId=FrmDraw[0]}
  [1353] = {x=-20.714, y=-5.465, z=137.434, rx=179.905, ry=0.202, rz=-129.709, fatherId=FrmDraw[0]}
  [1354] = {x=-20.58, y=-5.329, z=137.443, rx=179.916, ry=0.183, rz=-130.624, fatherId=FrmDraw[0]}
  [1355] = {x=-20.412, y=-5.209, z=137.454, rx=179.929, ry=0.16, rz=-131.8, fatherId=FrmDraw[0]}
  [1356] = {x=-20.238, y=-5.13, z=137.465, rx=179.941, ry=0.135, rz=-133.042, fatherId=FrmDraw[0]}
  [1357] = {x=-20.038, y=-5.079, z=137.477, rx=179.955, ry=0.107, rz=-134.489, fatherId=FrmDraw[0]}
  [1358] = {x=-19.84, y=-5.03, z=137.488, rx=179.967, ry=0.081, rz=-135.995, fatherId=FrmDraw[0]}
  [1359] = {x=-19.654, y=-4.971, z=137.499, rx=179.977, ry=0.059, rz=-137.491, fatherId=FrmDraw[0]}
  [1360] = {x=-19.523, y=-4.92, z=137.506, rx=179.983, ry=0.044, rz=-138.613, fatherId=FrmDraw[0]}
  [1361] = {x=-19.356, y=-4.845, z=137.515, rx=179.99, ry=0.029, rz=-140.122, fatherId=FrmDraw[0]}
  [1362] = {x=-19.201, y=-4.763, z=137.522, rx=179.994, ry=0.017, rz=-141.614, fatherId=FrmDraw[0]}
  [1363] = {x=-19.075, y=-4.687, z=137.529, rx=179.997, ry=0.008, rz=-142.904, fatherId=FrmDraw[0]}
  [1364] = {x=-18.966, y=-4.616, z=137.534, rx=179.999, ry=0.003, rz=-144.073, fatherId=FrmDraw[0]}
  [1365] = {x=-18.825, y=-4.514, z=137.54, rx=-179.999, ry=-0.003, rz=-145.667, fatherId=FrmDraw[0]}
  [1366] = {x=-18.699, y=-4.415, z=137.546, rx=-179.998, ry=-0.006, rz=-147.184, fatherId=FrmDraw[0]}
  [1367] = {x=-18.584, y=-4.317, z=137.55, rx=-179.998, ry=-0.008, rz=-148.636, fatherId=FrmDraw[0]}
  [1368] = {x=-18.479, y=-4.221, z=137.555, rx=-179.998, ry=-0.009, rz=-150.028, fatherId=FrmDraw[0]}
  [1369] = {x=-18.384, y=-4.125, z=137.558, rx=-179.998, ry=-0.008, rz=-151.368, fatherId=FrmDraw[0]}
  [1370] = {x=-18.296, y=-4.031, z=137.562, rx=-179.999, ry=-0.006, rz=-152.663, fatherId=FrmDraw[0]}
  [1371] = {x=-18.217, y=-3.938, z=137.564, rx=-179.999, ry=-0.003, rz=-153.918, fatherId=FrmDraw[0]}
  [1372] = {x=-18.143, y=-3.846, z=137.567, rx=180, ry=0.001, rz=-155.138, fatherId=FrmDraw[0]}
  [1373] = {x=-18.076, y=-3.756, z=137.569, rx=179.999, ry=0.006, rz=-156.327, fatherId=FrmDraw[0]}
  [1374] = {x=-18.015, y=-3.667, z=137.57, rx=179.998, ry=0.012, rz=-157.489, fatherId=FrmDraw[0]}
  [1375] = {x=-17.935, y=-3.54, z=137.572, rx=179.996, ry=0.022, rz=-159.14, fatherId=FrmDraw[0]}
  [1376] = {x=-17.874, y=-3.432, z=137.573, rx=179.994, ry=0.032, rz=-160.544, fatherId=FrmDraw[0]}
  [1377] = {x=-17.82, y=-3.327, z=137.574, rx=179.993, ry=0.043, rz=-161.908, fatherId=FrmDraw[0]}
  [1378] = {x=-17.765, y=-3.206, z=137.574, rx=179.992, ry=0.058, rz=-163.482, fatherId=FrmDraw[0]}
  [1379] = {x=-17.717, y=-3.09, z=137.574, rx=179.99, ry=0.074, rz=-165.047, fatherId=FrmDraw[0]}
  [1380] = {x=-17.675, y=-2.979, z=137.573, rx=179.989, ry=0.091, rz=-166.582, fatherId=FrmDraw[0]}
  [1381] = {x=-17.639, y=-2.875, z=137.572, rx=179.989, ry=0.108, rz=-168.101, fatherId=FrmDraw[0]}
  [1382] = {x=-17.607, y=-2.776, z=137.571, rx=179.988, ry=0.127, rz=-169.605, fatherId=FrmDraw[0]}
  [1383] = {x=-17.58, y=-2.682, z=137.569, rx=179.989, ry=0.145, rz=-171.097, fatherId=FrmDraw[0]}
  [1384] = {x=-17.556, y=-2.594, z=137.567, rx=179.989, ry=0.164, rz=-172.581, fatherId=FrmDraw[0]}
  [1385] = {x=-17.535, y=-2.512, z=137.565, rx=179.991, ry=0.183, rz=-174.058, fatherId=FrmDraw[0]}
  [1386] = {x=-17.517, y=-2.435, z=137.563, rx=179.992, ry=0.202, rz=-175.529, fatherId=FrmDraw[0]}
  [1387] = {x=-17.5, y=-2.363, z=137.56, rx=179.994, ry=0.221, rz=-176.997, fatherId=FrmDraw[0]}
  [1388] = {x=-17.486, y=-2.296, z=137.558, rx=179.997, ry=0.24, rz=-178.461, fatherId=FrmDraw[0]}
  [1389] = {x=-17.475, y=-2.208, z=137.554, rx=-179.999, ry=0.266, rz=179.622, fatherId=FrmDraw[0]}
  [1390] = {x=-17.472, y=-2.117, z=137.549, rx=-179.994, ry=0.295, rz=177.754, fatherId=FrmDraw[0]}
  [1391] = {x=-17.478, y=-2.026, z=137.544, rx=-179.988, ry=0.324, rz=175.928, fatherId=FrmDraw[0]}
  [1392] = {x=-17.493, y=-1.935, z=137.538, rx=-179.982, ry=0.356, rz=174.139, fatherId=FrmDraw[0]}
  [1393] = {x=-17.515, y=-1.842, z=137.532, rx=-179.974, ry=0.388, rz=172.388, fatherId=FrmDraw[0]}
  [1394] = {x=-17.547, y=-1.743, z=137.525, rx=-179.966, ry=0.423, rz=170.696, fatherId=FrmDraw[0]}
  [1395] = {x=-17.585, y=-1.639, z=137.518, rx=-179.956, ry=0.458, rz=169.059, fatherId=FrmDraw[0]}
  [1396] = {x=-17.628, y=-1.53, z=137.511, rx=-179.946, ry=0.492, rz=167.472, fatherId=FrmDraw[0]}
  [1397] = {x=-17.672, y=-1.415, z=137.504, rx=-179.935, ry=0.526, rz=165.93, fatherId=FrmDraw[0]}
  [1398] = {x=-17.716, y=-1.296, z=137.497, rx=-179.924, ry=0.557, rz=164.428, fatherId=FrmDraw[0]}
  [1399] = {x=-17.76, y=-1.173, z=137.49, rx=-179.912, ry=0.587, rz=162.962, fatherId=FrmDraw[0]}
  [1400] = {x=-17.805, y=-1.046, z=137.484, rx=-179.9, ry=0.615, rz=161.53, fatherId=FrmDraw[0]}
  [1401] = {x=-17.852, y=-0.915, z=137.477, rx=-179.888, ry=0.641, rz=160.13, fatherId=FrmDraw[0]}
  [1402] = {x=-17.902, y=-0.78, z=137.471, rx=-179.875, ry=0.668, rz=158.76, fatherId=FrmDraw[0]}
  [1403] = {x=-17.956, y=-0.641, z=137.464, rx=-179.861, ry=0.694, rz=157.419, fatherId=FrmDraw[0]}
  [1404] = {x=-18.015, y=-0.5, z=137.457, rx=-179.847, ry=0.721, rz=156.105, fatherId=FrmDraw[0]}
  [1405] = {x=-18.079, y=-0.356, z=137.45, rx=-179.833, ry=0.748, rz=154.817, fatherId=FrmDraw[0]}
  [1406] = {x=-18.15, y=-0.21, z=137.443, rx=-179.818, ry=0.776, rz=153.551, fatherId=FrmDraw[0]}
  [1407] = {x=-18.228, y=-0.062, z=137.435, rx=-179.801, ry=0.806, rz=152.308, fatherId=FrmDraw[0]}
  [1408] = {x=-18.313, y=0.084, z=137.427, rx=-179.784, ry=0.837, rz=151.073, fatherId=FrmDraw[0]}
  [1409] = {x=-18.403, y=0.228, z=137.419, rx=-179.766, ry=0.868, rz=149.833, fatherId=FrmDraw[0]}
  [1410] = {x=-18.498, y=0.367, z=137.41, rx=-179.747, ry=0.9, rz=148.587, fatherId=FrmDraw[0]}
  [1411] = {x=-18.598, y=0.503, z=137.401, rx=-179.727, ry=0.932, rz=147.332, fatherId=FrmDraw[0]}
  [1412] = {x=-18.701, y=0.635, z=137.392, rx=-179.706, ry=0.963, rz=146.068, fatherId=FrmDraw[0]}
  [1413] = {x=-18.807, y=0.763, z=137.383, rx=-179.685, ry=0.994, rz=144.794, fatherId=FrmDraw[0]}
  [1414] = {x=-18.915, y=0.887, z=137.374, rx=-179.662, ry=1.024, rz=143.506, fatherId=FrmDraw[0]}
  [1415] = {x=-19.026, y=1.008, z=137.365, rx=-179.639, ry=1.053, rz=142.205, fatherId=FrmDraw[0]}
  [1416] = {x=-19.137, y=1.124, z=137.357, rx=-179.616, ry=1.081, rz=140.889, fatherId=FrmDraw[0]}
  [1417] = {x=-19.249, y=1.237, z=137.348, rx=-179.592, ry=1.107, rz=139.555, fatherId=FrmDraw[0]}
  [1418] = {x=-19.363, y=1.354, z=137.34, rx=-179.568, ry=1.133, rz=138.239, fatherId=FrmDraw[0]}
  [1419] = {x=-19.421, y=1.416, z=137.335, rx=-179.556, ry=1.146, rz=137.6, fatherId=FrmDraw[0]}
  [1420] = {x=-19.51, y=1.514, z=137.329, rx=-179.537, ry=1.165, rz=136.666, fatherId=FrmDraw[0]}
  [1421] = {x=-19.631, y=1.655, z=137.32, rx=-179.512, ry=1.192, rz=135.467, fatherId=FrmDraw[0]}
  [1422] = {x=-19.755, y=1.807, z=137.311, rx=-179.486, ry=1.219, rz=134.32, fatherId=FrmDraw[0]}
  [1423] = {x=-19.881, y=1.971, z=137.302, rx=-179.461, ry=1.247, rz=133.226, fatherId=FrmDraw[0]}
  [1424] = {x=-20.01, y=2.147, z=137.293, rx=-179.435, ry=1.275, rz=132.185, fatherId=FrmDraw[0]}
  [1425] = {x=-20.141, y=2.336, z=137.284, rx=-179.409, ry=1.304, rz=131.198, fatherId=FrmDraw[0]}
  [1426] = {x=-20.273, y=2.537, z=137.275, rx=-179.382, ry=1.332, rz=130.265, fatherId=FrmDraw[0]}
  [1427] = {x=-20.407, y=2.752, z=137.266, rx=-179.356, ry=1.362, rz=129.386, fatherId=FrmDraw[0]}
  [1428] = {x=-20.54, y=2.977, z=137.257, rx=-179.33, ry=1.39, rz=128.546, fatherId=FrmDraw[0]}
  [1429] = {x=-20.674, y=3.204, z=137.249, rx=-179.304, ry=1.417, rz=127.703, fatherId=FrmDraw[0]}
  [1430] = {x=-20.808, y=3.432, z=137.241, rx=-179.279, ry=1.442, rz=126.855, fatherId=FrmDraw[0]}
  [1431] = {x=-20.942, y=3.661, z=137.234, rx=-179.254, ry=1.465, rz=126.001, fatherId=FrmDraw[0]}
  [1432] = {x=-21.078, y=3.892, z=137.226, rx=-179.228, ry=1.487, rz=125.14, fatherId=FrmDraw[0]}
  [1433] = {x=-21.215, y=4.124, z=137.22, rx=-179.203, ry=1.507, rz=124.272, fatherId=FrmDraw[0]}
  [1434] = {x=-21.354, y=4.357, z=137.213, rx=-179.179, ry=1.525, rz=123.397, fatherId=FrmDraw[0]}
  [1435] = {x=-21.496, y=4.59, z=137.207, rx=-179.154, ry=1.543, rz=122.515, fatherId=FrmDraw[0]}
  [1436] = {x=-21.604, y=4.766, z=137.202, rx=-179.135, ry=1.555, rz=121.847, fatherId=FrmDraw[0]}
  [1437] = {x=-21.742, y=4.989, z=137.197, rx=-179.112, ry=1.57, rz=121.005, fatherId=FrmDraw[0]}
  [1438] = {x=-21.885, y=5.231, z=137.191, rx=-179.087, ry=1.586, rz=120.185, fatherId=FrmDraw[0]}
  [1439] = {x=-22.007, y=5.452, z=137.186, rx=-179.067, ry=1.602, rz=119.531, fatherId=FrmDraw[0]}
  [1440] = {x=-22.108, y=5.646, z=137.182, rx=-179.049, ry=1.615, rz=119.021, fatherId=FrmDraw[0]}
  [1441] = {x=-22.246, y=5.933, z=137.177, rx=-179.025, ry=1.633, rz=118.362, fatherId=FrmDraw[0]}
  [1442] = {x=-22.361, y=6.195, z=137.173, rx=-179.005, ry=1.65, rz=117.85, fatherId=FrmDraw[0]}
  [1443] = {x=-22.45, y=6.415, z=137.169, rx=-178.99, ry=1.664, rz=117.476, fatherId=FrmDraw[0]}
  [1444] = {x=-22.557, y=6.703, z=137.166, rx=-178.971, ry=1.681, rz=117.055, fatherId=FrmDraw[0]}
  [1445] = {x=-22.639, y=6.945, z=137.163, rx=-178.957, ry=1.694, rz=116.754, fatherId=FrmDraw[0]}
  [1446] = {x=-22.734, y=7.263, z=137.16, rx=-178.939, ry=1.711, rz=116.425, fatherId=FrmDraw[0]}
  [1447] = {x=-22.804, y=7.529, z=137.158, rx=-178.927, ry=1.724, rz=116.2, fatherId=FrmDraw[0]}
  [1448] = {x=-22.886, y=7.872, z=137.156, rx=-178.912, ry=1.74, rz=115.946, fatherId=FrmDraw[0]}
  [1449] = {x=-22.949, y=8.15, z=137.156, rx=-178.901, ry=1.75, rz=115.747, fatherId=FrmDraw[0]}
  [1450] = {x=-23.024, y=8.502, z=137.155, rx=-178.888, ry=1.762, rz=115.501, fatherId=FrmDraw[0]}
  [1451] = {x=-23.082, y=8.787, z=137.154, rx=-178.879, ry=1.77, rz=115.308, fatherId=FrmDraw[0]}
  [1452] = {x=-23.152, y=9.148, z=137.155, rx=-178.868, ry=1.779, rz=115.07, fatherId=FrmDraw[0]}
  [1453] = {x=-23.206, y=9.439, z=137.155, rx=-178.86, ry=1.786, rz=114.884, fatherId=FrmDraw[0]}
  [1454] = {x=-23.273, y=9.806, z=137.155, rx=-178.85, ry=1.793, rz=114.655, fatherId=FrmDraw[0]}
  [1455] = {x=-23.326, y=10.102, z=137.156, rx=-178.843, ry=1.799, rz=114.475, fatherId=FrmDraw[0]}
  [1456] = {x=-23.392, y=10.475, z=137.157, rx=-178.833, ry=1.805, rz=114.255, fatherId=FrmDraw[0]}
  [1457] = {x=-23.444, y=10.776, z=137.158, rx=-178.826, ry=1.81, rz=114.082, fatherId=FrmDraw[0]}
  [1458] = {x=-23.511, y=11.153, z=137.159, rx=-178.817, ry=1.817, rz=113.871, fatherId=FrmDraw[0]}
  [1459] = {x=-23.565, y=11.455, z=137.16, rx=-178.81, ry=1.822, rz=113.703, fatherId=FrmDraw[0]}
  [1460] = {x=-23.635, y=11.834, z=137.161, rx=-178.801, ry=1.829, rz=113.492, fatherId=FrmDraw[0]}
  [1461] = {x=-23.693, y=12.137, z=137.162, rx=-178.793, ry=1.835, rz=113.323, fatherId=FrmDraw[0]}
  [1462] = {x=-23.766, y=12.516, z=137.163, rx=-178.783, ry=1.842, rz=113.111, fatherId=FrmDraw[0]}
  [1463] = {x=-23.826, y=12.821, z=137.164, rx=-178.776, ry=1.848, rz=112.94, fatherId=FrmDraw[0]}
  [1464] = {x=-23.903, y=13.201, z=137.166, rx=-178.766, ry=1.855, rz=112.727, fatherId=FrmDraw[0]}
  [1465] = {x=-23.965, y=13.507, z=137.167, rx=-178.758, ry=1.861, rz=112.555, fatherId=FrmDraw[0]}
  [1466] = {x=-24.045, y=13.889, z=137.169, rx=-178.748, ry=1.868, rz=112.34, fatherId=FrmDraw[0]}
  [1467] = {x=-24.11, y=14.195, z=137.17, rx=-178.74, ry=1.873, rz=112.167, fatherId=FrmDraw[0]}
  [1468] = {x=-24.192, y=14.58, z=137.172, rx=-178.731, ry=1.88, rz=111.95, fatherId=FrmDraw[0]}
  [1469] = {x=-24.258, y=14.888, z=137.173, rx=-178.723, ry=1.885, rz=111.776, fatherId=FrmDraw[0]}
  [1470] = {x=-24.342, y=15.274, z=137.175, rx=-178.713, ry=1.891, rz=111.557, fatherId=FrmDraw[0]}
  [1471] = {x=-24.41, y=15.584, z=137.176, rx=-178.706, ry=1.896, rz=111.382, fatherId=FrmDraw[0]}
  [1472] = {x=-24.496, y=15.974, z=137.179, rx=-178.697, ry=1.902, rz=111.161, fatherId=FrmDraw[0]}
  [1473] = {x=-24.565, y=16.286, z=137.18, rx=-178.69, ry=1.906, rz=110.985, fatherId=FrmDraw[0]}
  [1474] = {x=-24.652, y=16.678, z=137.183, rx=-178.681, ry=1.91, rz=110.762, fatherId=FrmDraw[0]}
  [1475] = {x=-24.722, y=16.993, z=137.185, rx=-178.675, ry=1.914, rz=110.584, fatherId=FrmDraw[0]}
  [1476] = {x=-24.809, y=17.388, z=137.187, rx=-178.667, ry=1.917, rz=110.36, fatherId=FrmDraw[0]}
  [1477] = {x=-24.88, y=17.706, z=137.189, rx=-178.661, ry=1.919, rz=110.18, fatherId=FrmDraw[0]}
  [1478] = {x=-24.968, y=18.106, z=137.192, rx=-178.654, ry=1.921, rz=109.954, fatherId=FrmDraw[0]}
  [1479] = {x=-25.038, y=18.427, z=137.195, rx=-178.648, ry=1.922, rz=109.773, fatherId=FrmDraw[0]}
  [1480] = {x=-25.128, y=18.829, z=137.198, rx=-178.642, ry=1.923, rz=109.542, fatherId=FrmDraw[0]}
  [1481] = {x=-25.2, y=19.152, z=137.2, rx=-178.637, ry=1.923, rz=109.355, fatherId=FrmDraw[0]}
  [1482] = {x=-25.293, y=19.556, z=137.203, rx=-178.632, ry=1.922, rz=109.117, fatherId=FrmDraw[0]}
  [1483] = {x=-25.37, y=19.879, z=137.206, rx=-178.627, ry=1.922, rz=108.924, fatherId=FrmDraw[0]}
  [1484] = {x=-25.47, y=20.283, z=137.209, rx=-178.621, ry=1.922, rz=108.679, fatherId=FrmDraw[0]}
  [1485] = {x=-25.553, y=20.605, z=137.211, rx=-178.616, ry=1.922, rz=108.479, fatherId=FrmDraw[0]}
  [1486] = {x=-25.662, y=21.007, z=137.214, rx=-178.608, ry=1.923, rz=108.226, fatherId=FrmDraw[0]}
  [1487] = {x=-25.753, y=21.327, z=137.217, rx=-178.602, ry=1.925, rz=108.02, fatherId=FrmDraw[0]}
  [1488] = {x=-25.874, y=21.725, z=137.219, rx=-178.593, ry=1.928, rz=107.758, fatherId=FrmDraw[0]}
  [1489] = {x=-25.975, y=22.042, z=137.221, rx=-178.585, ry=1.932, rz=107.55, fatherId=FrmDraw[0]}
  [1490] = {x=-26.094, y=22.447, z=137.224, rx=-178.574, ry=1.938, rz=107.318, fatherId=FrmDraw[0]}
  [1491] = {x=-26.198, y=22.85, z=137.228, rx=-178.564, ry=1.945, rz=107.127, fatherId=FrmDraw[0]}
  [1492] = {x=-26.276, y=23.208, z=137.231, rx=-178.556, ry=1.951, rz=106.991, fatherId=FrmDraw[0]}
  [1493] = {x=-26.349, y=23.637, z=137.235, rx=-178.548, ry=1.957, rz=106.865, fatherId=FrmDraw[0]}
  [1494] = {x=-26.395, y=24.021, z=137.24, rx=-178.543, ry=1.961, rz=106.784, fatherId=FrmDraw[0]}
  [1495] = {x=-26.426, y=24.484, z=137.245, rx=-178.541, ry=1.961, rz=106.722, fatherId=FrmDraw[0]}
  [1496] = {x=-26.431, y=24.9, z=137.251, rx=-178.543, ry=1.958, rz=106.697, fatherId=FrmDraw[0]}
  [1497] = {x=-26.408, y=25.404, z=137.257, rx=-178.55, ry=1.949, rz=106.7, fatherId=FrmDraw[0]}
  [1498] = {x=-26.47, y=25.781, z=137.261, rx=-178.558, ry=1.931, rz=106.496, fatherId=FrmDraw[0]}
  [1499] = {x=-26.46, y=25.786, z=137.678, rx=-178.559, ry=1.931, rz=106.513, fatherId=FrmDraw[0]}
public pointRx shere = {x=978.504226, y=-109.919125, z=104.826018, rx=-0.09799, ry=179.816018, rz=56.09787, shoulder=lefty, elbow=epositive, wrist=wpositive, fatherId=world[0]}
public sio sSocketout = {link=Socket\CClient}
public string l_sString[6] = "978.504,-109.919,104.826,"
string sString[1500]
  [0] = "-21.496000,-9.920000,104.826000,179.902000,0.184000,-123.901000,"
  [1] = "-21.406000,-9.571000,104.833000,179.906000,0.177000,-124.352000,"
  [2] = "-21.327000,-9.235000,104.840000,179.910000,0.172000,-124.769000,"
  [3] = "-21.269000,-8.967000,104.845000,179.913000,0.168000,-125.087000,"
  [4] = "-21.197000,-8.609000,104.852000,179.915000,0.164000,-125.501000,"
  [5] = "-21.125000,-8.284000,104.858000,179.919000,0.159000,-125.914000,"
  [6] = "-21.063000,-8.029000,104.863000,179.922000,0.154000,-126.277000,"
  [7] = "-20.979000,-7.711000,104.871000,179.927000,0.146000,-126.778000,"
  [8] = "-20.888000,-7.402000,104.879000,179.933000,0.136000,-127.324000,"
  [9] = "-20.796000,-7.121000,104.886000,179.939000,0.125000,-127.880000,"
  [10] = "-20.693000,-6.864000,104.895000,179.946000,0.112000,-128.514000,"
  [11] = "-20.565000,-6.611000,104.905000,179.956000,0.094000,-129.312000,"
  [12] = "-20.433000,-6.398000,104.914000,179.965000,0.076000,-130.171000,"
  [13] = "-20.305000,-6.222000,104.923000,179.973000,0.059000,-131.051000,"
  [14] = "-20.156000,-6.043000,104.933000,179.981000,0.042000,-132.148000,"
  [15] = "-20.038000,-5.901000,104.940000,179.986000,0.032000,-133.098000,"
  [16] = "-19.899000,-5.734000,104.948000,179.990000,0.023000,-134.309000,"
  [17] = "-19.764000,-5.576000,104.955000,179.993000,0.017000,-135.558000,"
  [18] = "-19.634000,-5.431000,104.961000,179.995000,0.013000,-136.824000,"
  [19] = "-19.514000,-5.306000,104.967000,179.997000,0.008000,-138.020000,"
  [20] = "-19.402000,-5.193000,104.973000,179.998000,0.005000,-139.156000,"
  [21] = "-19.268000,-5.059000,104.979000,-180.000000,-0.000000,-140.558000,"
  [22] = "-19.155000,-4.950000,104.985000,-179.999000,-0.004000,-141.768000,"
  [23] = "-19.052000,-4.852000,104.990000,-179.997000,-0.008000,-142.893000,"
  [24] = "-18.935000,-4.744000,104.995000,-179.996000,-0.013000,-144.181000,"
  [25] = "-18.824000,-4.636000,105.001000,-179.995000,-0.017000,-145.451000,"
  [26] = "-18.703000,-4.509000,105.006000,-179.994000,-0.021000,-146.890000,"
  [27] = "-18.592000,-4.383000,105.011000,-179.993000,-0.023000,-148.260000,"
  [28] = "-18.492000,-4.260000,105.016000,-179.993000,-0.024000,-149.572000,"
  [29] = "-18.401000,-4.137000,105.020000,-179.994000,-0.023000,-150.833000,"
  [30] = "-18.318000,-4.016000,105.023000,-179.995000,-0.022000,-152.050000,"
  [31] = "-18.223000,-3.864000,105.027000,-179.996000,-0.017000,-153.555000,"
  [32] = "-18.157000,-3.747000,105.029000,-179.997000,-0.012000,-154.683000,"
  [33] = "-18.097000,-3.632000,105.031000,-179.999000,-0.006000,-155.782000,"
  [34] = "-18.044000,-3.519000,105.032000,180.000000,0.001000,-156.854000,"
  [35] = "-17.996000,-3.408000,105.033000,179.998000,0.010000,-157.905000,"
  [36] = "-17.952000,-3.300000,105.034000,179.996000,0.019000,-158.942000,"
  [37] = "-17.893000,-3.145000,105.035000,179.994000,0.034000,-160.472000,"
  [38] = "-17.842000,-2.998000,105.035000,179.992000,0.050000,-161.989000,"
  [39] = "-17.798000,-2.858000,105.034000,179.990000,0.068000,-163.483000,"
  [40] = "-17.759000,-2.726000,105.033000,179.989000,0.087000,-164.962000,"
  [41] = "-17.726000,-2.601000,105.032000,179.987000,0.106000,-166.428000,"
  [42] = "-17.699000,-2.483000,105.030000,179.987000,0.127000,-167.883000,"
  [43] = "-17.676000,-2.372000,105.028000,179.986000,0.148000,-169.329000,"
  [44] = "-17.657000,-2.266000,105.026000,179.986000,0.170000,-170.767000,"
  [45] = "-17.643000,-2.167000,105.023000,179.987000,0.193000,-172.197000,"
  [46] = "-17.635000,-2.070000,105.020000,179.988000,0.217000,-173.604000,"
  [47] = "-17.631000,-1.974000,105.016000,179.989000,0.242000,-174.986000,"
  [48] = "-17.632000,-1.879000,105.012000,179.991000,0.268000,-176.347000,"
  [49] = "-17.636000,-1.787000,105.008000,179.994000,0.293000,-177.689000,"
  [50] = "-17.643000,-1.696000,105.004000,179.997000,0.319000,-179.015000,"
  [51] = "-17.654000,-1.579000,104.998000,-179.998000,0.353000,179.235000,"
  [52] = "-17.666000,-1.469000,104.993000,-179.992000,0.384000,177.491000,"
  [53] = "-17.679000,-1.366000,104.987000,-179.985000,0.414000,175.749000,"
  [54] = "-17.691000,-1.271000,104.982000,-179.977000,0.442000,174.006000,"
  [55] = "-17.704000,-1.183000,104.977000,-179.968000,0.469000,172.258000,"
  [56] = "-17.721000,-1.092000,104.972000,-179.959000,0.496000,170.546000,"
  [57] = "-17.744000,-0.993000,104.966000,-179.949000,0.523000,168.902000,"
  [58] = "-17.774000,-0.886000,104.960000,-179.939000,0.552000,167.322000,"
  [59] = "-17.809000,-0.770000,104.954000,-179.928000,0.582000,165.802000,"
  [60] = "-17.851000,-0.646000,104.947000,-179.916000,0.612000,164.339000,"
  [61] = "-17.898000,-0.515000,104.940000,-179.903000,0.644000,162.930000,"
  [62] = "-17.951000,-0.376000,104.932000,-179.890000,0.676000,161.572000,"
  [63] = "-18.009000,-0.231000,104.925000,-179.877000,0.708000,160.261000,"
  [64] = "-18.071000,-0.079000,104.917000,-179.863000,0.741000,158.995000,"
  [65] = "-18.137000,0.079000,104.908000,-179.848000,0.775000,157.770000,"
  [66] = "-18.207000,0.239000,104.900000,-179.833000,0.807000,156.562000,"
  [67] = "-18.277000,0.395000,104.892000,-179.817000,0.839000,155.349000,"
  [68] = "-18.350000,0.548000,104.885000,-179.800000,0.869000,154.132000,"
  [69] = "-18.426000,0.698000,104.877000,-179.784000,0.898000,152.908000,"
  [70] = "-18.504000,0.844000,104.869000,-179.766000,0.927000,151.676000,"
  [71] = "-18.584000,0.987000,104.861000,-179.748000,0.955000,150.435000,"
  [72] = "-18.668000,1.126000,104.854000,-179.729000,0.983000,149.184000,"
  [73] = "-18.756000,1.261000,104.846000,-179.710000,1.010000,147.922000,"
  [74] = "-18.847000,1.391000,104.838000,-179.689000,1.037000,146.647000,"
  [75] = "-18.943000,1.517000,104.830000,-179.668000,1.064000,145.357000,"
  [76] = "-19.043000,1.640000,104.821000,-179.646000,1.092000,144.066000,"
  [77] = "-19.149000,1.767000,104.812000,-179.623000,1.121000,142.804000,"
  [78] = "-19.258000,1.900000,104.803000,-179.599000,1.151000,141.570000,"
  [79] = "-19.315000,1.968000,104.799000,-179.587000,1.166000,140.964000,"
  [80] = "-19.401000,2.072000,104.792000,-179.568000,1.190000,140.069000,"
  [81] = "-19.518000,2.217000,104.782000,-179.542000,1.221000,138.900000,"
  [82] = "-19.638000,2.368000,104.772000,-179.516000,1.252000,137.760000,"
  [83] = "-19.759000,2.525000,104.763000,-179.490000,1.282000,136.648000,"
  [84] = "-19.880000,2.688000,104.754000,-179.464000,1.312000,135.564000,"
  [85] = "-20.001000,2.860000,104.745000,-179.438000,1.340000,134.508000,"
  [86] = "-20.122000,3.039000,104.736000,-179.412000,1.367000,133.478000,"
  [87] = "-20.240000,3.225000,104.728000,-179.387000,1.391000,132.471000,"
  [88] = "-20.358000,3.418000,104.721000,-179.363000,1.413000,131.482000,"
  [89] = "-20.475000,3.617000,104.714000,-179.339000,1.434000,130.511000,"
  [90] = "-20.592000,3.823000,104.707000,-179.316000,1.453000,129.559000,"
  [91] = "-20.710000,4.035000,104.701000,-179.293000,1.471000,128.624000,"
  [92] = "-20.823000,4.242000,104.695000,-179.271000,1.487000,127.752000,"
  [93] = "-20.943000,4.465000,104.689000,-179.248000,1.504000,126.851000,"
  [94] = "-21.066000,4.694000,104.683000,-179.224000,1.521000,125.967000,"
  [95] = "-21.192000,4.928000,104.677000,-179.201000,1.538000,125.099000,"
  [96] = "-21.321000,5.168000,104.670000,-179.177000,1.556000,124.249000,"
  [97] = "-21.453000,5.415000,104.664000,-179.153000,1.575000,123.427000,"
  [98] = "-21.587000,5.671000,104.658000,-179.128000,1.594000,122.636000,"
  [99] = "-21.722000,5.937000,104.652000,-179.103000,1.615000,121.878000,"
  [100] = "-21.857000,6.213000,104.646000,-179.078000,1.635000,121.155000,"
  [101] = "-21.990000,6.500000,104.640000,-179.053000,1.655000,120.468000,"
  [102] = "-22.118000,6.791000,104.635000,-179.030000,1.674000,119.831000,"
  [103] = "-22.226000,7.051000,104.631000,-179.011000,1.690000,119.312000,"
  [104] = "-22.313000,7.274000,104.628000,-178.995000,1.702000,118.900000,"
  [105] = "-22.431000,7.598000,104.624000,-178.975000,1.718000,118.352000,"
  [106] = "-22.528000,7.887000,104.622000,-178.958000,1.731000,117.910000,"
  [107] = "-22.602000,8.124000,104.620000,-178.946000,1.740000,117.572000,"
  [108] = "-22.692000,8.429000,104.618000,-178.931000,1.750000,117.171000,"
  [109] = "-22.762000,8.680000,104.617000,-178.920000,1.757000,116.866000,"
  [110] = "-22.845000,9.001000,104.617000,-178.908000,1.765000,116.506000,"
  [111] = "-22.909000,9.265000,104.616000,-178.898000,1.772000,116.235000,"
  [112] = "-22.985000,9.602000,104.616000,-178.887000,1.779000,115.918000,"
  [113] = "-23.044000,9.878000,104.616000,-178.878000,1.784000,115.682000,"
  [114] = "-23.114000,10.232000,104.616000,-178.868000,1.791000,115.409000,"
  [115] = "-23.168000,10.520000,104.617000,-178.860000,1.797000,115.209000,"
  [116] = "-23.231000,10.889000,104.617000,-178.850000,1.804000,114.981000,"
  [117] = "-23.280000,11.188000,104.618000,-178.843000,1.809000,114.813000,"
  [118] = "-23.341000,11.564000,104.619000,-178.834000,1.816000,114.603000,"
  [119] = "-23.391000,11.865000,104.620000,-178.827000,1.821000,114.433000,"
  [120] = "-23.455000,12.243000,104.621000,-178.819000,1.827000,114.218000,"
  [121] = "-23.507000,12.545000,104.623000,-178.812000,1.831000,114.045000,"
  [122] = "-23.573000,12.924000,104.624000,-178.804000,1.836000,113.827000,"
  [123] = "-23.626000,13.227000,104.625000,-178.797000,1.840000,113.651000,"
  [124] = "-23.695000,13.607000,104.627000,-178.789000,1.844000,113.428000,"
  [125] = "-23.751000,13.912000,104.628000,-178.783000,1.847000,113.248000,"
  [126] = "-23.823000,14.293000,104.630000,-178.775000,1.851000,113.022000,"
  [127] = "-23.882000,14.598000,104.632000,-178.769000,1.854000,112.839000,"
  [128] = "-23.957000,14.981000,104.634000,-178.761000,1.858000,112.607000,"
  [129] = "-24.019000,15.287000,104.635000,-178.755000,1.861000,112.421000,"
  [130] = "-24.098000,15.670000,104.637000,-178.747000,1.864000,112.186000,"
  [131] = "-24.163000,15.977000,104.639000,-178.741000,1.867000,111.995000,"
  [132] = "-24.246000,16.361000,104.641000,-178.733000,1.870000,111.755000,"
  [133] = "-24.315000,16.668000,104.642000,-178.726000,1.873000,111.562000,"
  [134] = "-24.403000,17.053000,104.645000,-178.718000,1.877000,111.317000,"
  [135] = "-24.476000,17.360000,104.646000,-178.711000,1.880000,111.120000,"
  [136] = "-24.570000,17.745000,104.648000,-178.702000,1.883000,110.870000,"
  [137] = "-24.647000,18.053000,104.650000,-178.695000,1.887000,110.669000,"
  [138] = "-24.746000,18.438000,104.652000,-178.686000,1.891000,110.415000,"
  [139] = "-24.827000,18.746000,104.654000,-178.678000,1.895000,110.213000,"
  [140] = "-24.929000,19.134000,104.656000,-178.669000,1.900000,109.963000,"
  [141] = "-25.011000,19.446000,104.657000,-178.661000,1.904000,109.767000,"
  [142] = "-25.114000,19.839000,104.660000,-178.651000,1.909000,109.526000,"
  [143] = "-25.196000,20.155000,104.662000,-178.643000,1.914000,109.336000,"
  [144] = "-25.298000,20.553000,104.664000,-178.634000,1.918000,109.102000,"
  [145] = "-25.378000,20.875000,104.667000,-178.627000,1.922000,108.919000,"
  [146] = "-25.478000,21.279000,104.670000,-178.619000,1.925000,108.693000,"
  [147] = "-25.556000,21.606000,104.672000,-178.613000,1.928000,108.516000,"
  [148] = "-25.651000,22.019000,104.675000,-178.606000,1.929000,108.299000,"
  [149] = "-25.727000,22.351000,104.678000,-178.601000,1.930000,108.126000,"
  [150] = "-25.823000,22.767000,104.682000,-178.596000,1.929000,107.903000,"
  [151] = "-25.901000,23.101000,104.684000,-178.592000,1.928000,107.720000,"
  [152] = "-26.003000,23.518000,104.688000,-178.588000,1.925000,107.485000,"
  [153] = "-26.087000,23.851000,104.691000,-178.585000,1.923000,107.292000,"
  [154] = "-26.197000,24.266000,104.694000,-178.580000,1.920000,107.045000,"
  [155] = "-26.310000,24.666000,104.697000,-178.575000,1.918000,106.799000,"
  [156] = "-26.411000,25.010000,104.700000,-178.571000,1.917000,106.581000,"
  [157] = "-26.536000,25.406000,104.703000,-178.564000,1.916000,106.322000,"
  [158] = "-26.745000,25.675000,104.703000,-178.557000,1.911000,105.881000,"
  [159] = "-26.744000,25.675000,105.202000,-178.556000,1.913000,105.887000,"
  [160] = "-26.743000,25.675000,105.702000,-178.555000,1.914000,105.893000,"
  [161] = "-26.743000,25.675000,106.101000,-178.554000,1.915000,105.898000,"
  [162] = "-26.742000,25.675000,106.501000,-178.554000,1.916000,105.903000,"
  [163] = "-26.742000,25.675000,106.740000,-178.553000,1.917000,105.906000,"
  [164] = "-26.742000,25.675000,107.100000,-178.553000,1.918000,105.910000,"
  [165] = "-26.741000,25.674000,107.578000,-178.552000,1.919000,105.916000,"
  [166] = "-26.741000,25.674000,108.029000,-178.551000,1.920000,105.921000,"
  [167] = "-26.740000,25.674000,108.403000,-178.550000,1.921000,105.926000,"
  [168] = "-26.740000,25.674000,108.777000,-178.550000,1.922000,105.930000,"
  [169] = "-26.577000,25.370000,108.776000,-178.554000,1.929000,106.286000,"
  [170] = "-26.456000,24.972000,108.772000,-178.558000,1.932000,106.549000,"
  [171] = "-26.355000,24.627000,108.770000,-178.562000,1.935000,106.769000,"
  [172] = "-26.243000,24.227000,108.766000,-178.566000,1.938000,107.016000,"
  [173] = "-26.132000,23.812000,108.763000,-178.572000,1.940000,107.263000,"
  [174] = "-26.046000,23.480000,108.760000,-178.576000,1.941000,107.454000,"
  [175] = "-25.943000,23.065000,108.757000,-178.581000,1.941000,107.685000,"
  [176] = "-25.863000,22.732000,108.754000,-178.586000,1.941000,107.863000,"
  [177] = "-25.766000,22.316000,108.750000,-178.592000,1.940000,108.078000,"
  [178] = "-25.691000,21.983000,108.748000,-178.598000,1.938000,108.244000,"
  [179] = "-25.597000,21.568000,108.744000,-178.605000,1.936000,108.453000,"
  [180] = "-25.521000,21.240000,108.742000,-178.611000,1.934000,108.625000,"
  [181] = "-25.424000,20.833000,108.739000,-178.619000,1.930000,108.844000,"
  [182] = "-25.346000,20.510000,108.736000,-178.626000,1.927000,109.024000,"
  [183] = "-25.247000,20.109000,108.733000,-178.634000,1.924000,109.254000,"
  [184] = "-25.167000,19.791000,108.731000,-178.641000,1.921000,109.442000,"
  [185] = "-25.067000,19.396000,108.729000,-178.650000,1.917000,109.683000,"
  [186] = "-24.987000,19.083000,108.727000,-178.657000,1.914000,109.879000,"
  [187] = "-24.886000,18.694000,108.724000,-178.666000,1.910000,110.129000,"
  [188] = "-24.806000,18.384000,108.723000,-178.673000,1.907000,110.333000,"
  [189] = "-24.707000,17.999000,108.720000,-178.681000,1.904000,110.589000,"
  [190] = "-24.630000,17.691000,108.719000,-178.688000,1.901000,110.792000,"
  [191] = "-24.537000,17.306000,108.716000,-178.697000,1.898000,111.043000,"
  [192] = "-24.464000,16.999000,108.715000,-178.703000,1.895000,111.241000,"
  [193] = "-24.375000,16.615000,108.712000,-178.712000,1.892000,111.486000,"
  [194] = "-24.305000,16.308000,108.711000,-178.718000,1.889000,111.681000,"
  [195] = "-24.221000,15.924000,108.709000,-178.726000,1.885000,111.921000,"
  [196] = "-24.155000,15.618000,108.707000,-178.733000,1.882000,112.111000,"
  [197] = "-24.074000,15.236000,108.705000,-178.741000,1.878000,112.345000,"
  [198] = "-24.011000,14.930000,108.704000,-178.748000,1.875000,112.531000,"
  [199] = "-23.935000,14.548000,108.702000,-178.756000,1.871000,112.761000,"
  [200] = "-23.875000,14.243000,108.700000,-178.763000,1.867000,112.943000,"
  [201] = "-23.802000,13.863000,108.698000,-178.771000,1.862000,113.169000,"
  [202] = "-23.744000,13.559000,108.697000,-178.778000,1.859000,113.347000,"
  [203] = "-23.674000,13.179000,108.696000,-178.786000,1.853000,113.567000,"
  [204] = "-23.620000,12.876000,108.694000,-178.793000,1.849000,113.741000,"
  [205] = "-23.552000,12.497000,108.693000,-178.802000,1.843000,113.957000,"
  [206] = "-23.500000,12.195000,108.692000,-178.809000,1.839000,114.128000,"
  [207] = "-23.435000,11.818000,108.690000,-178.818000,1.832000,114.339000,"
  [208] = "-23.385000,11.516000,108.689000,-178.825000,1.827000,114.506000,"
  [209] = "-23.323000,11.140000,108.688000,-178.834000,1.820000,114.713000,"
  [210] = "-23.274000,10.840000,108.688000,-178.841000,1.814000,114.879000,"
  [211] = "-23.210000,10.471000,108.687000,-178.851000,1.807000,115.105000,"
  [212] = "-23.156000,10.182000,108.686000,-178.859000,1.802000,115.303000,"
  [213] = "-23.086000,9.828000,108.686000,-178.869000,1.795000,115.571000,"
  [214] = "-23.028000,9.550000,108.686000,-178.878000,1.789000,115.802000,"
  [215] = "-22.952000,9.210000,108.686000,-178.889000,1.782000,116.110000,"
  [216] = "-22.889000,8.945000,108.686000,-178.899000,1.775000,116.373000,"
  [217] = "-22.806000,8.621000,108.687000,-178.912000,1.766000,116.721000,"
  [218] = "-22.737000,8.368000,108.688000,-178.923000,1.759000,117.016000,"
  [219] = "-22.656000,8.090000,108.690000,-178.936000,1.749000,117.363000,"
  [220] = "-22.572000,7.820000,108.692000,-178.950000,1.738000,117.728000,"
  [221] = "-22.475000,7.528000,108.695000,-178.967000,1.724000,118.152000,"
  [222] = "-22.355000,7.201000,108.699000,-178.988000,1.706000,118.682000,"
  [223] = "-22.267000,6.976000,108.702000,-179.004000,1.693000,119.085000,"
  [224] = "-22.157000,6.715000,108.706000,-179.024000,1.676000,119.593000,"
  [225] = "-22.026000,6.423000,108.711000,-179.048000,1.656000,120.221000,"
  [226] = "-21.890000,6.136000,108.717000,-179.074000,1.634000,120.903000,"
  [227] = "-21.752000,5.860000,108.724000,-179.099000,1.613000,121.625000,"
  [228] = "-21.615000,5.596000,108.730000,-179.124000,1.592000,122.385000,"
  [229] = "-21.478000,5.341000,108.736000,-179.150000,1.572000,123.182000,"
  [230] = "-21.344000,5.097000,108.742000,-179.174000,1.553000,124.013000,"
  [231] = "-21.213000,4.859000,108.748000,-179.198000,1.536000,124.871000,"
  [232] = "-21.087000,4.625000,108.754000,-179.221000,1.519000,125.743000,"
  [233] = "-20.964000,4.397000,108.760000,-179.244000,1.503000,126.629000,"
  [234] = "-20.843000,4.173000,108.766000,-179.267000,1.486000,127.529000,"
  [235] = "-20.730000,3.965000,108.772000,-179.289000,1.470000,128.397000,"
  [236] = "-20.612000,3.751000,108.778000,-179.312000,1.452000,129.324000,"
  [237] = "-20.495000,3.543000,108.785000,-179.336000,1.433000,130.267000,"
  [238] = "-20.377000,3.341000,108.792000,-179.360000,1.413000,131.224000,"
  [239] = "-20.259000,3.144000,108.800000,-179.384000,1.390000,132.196000,"
  [240] = "-20.139000,2.954000,108.808000,-179.409000,1.365000,133.183000,"
  [241] = "-20.017000,2.772000,108.817000,-179.435000,1.337000,134.197000,"
  [242] = "-19.894000,2.599000,108.826000,-179.461000,1.309000,135.242000,"
  [243] = "-19.772000,2.434000,108.835000,-179.487000,1.279000,136.319000,"
  [244] = "-19.650000,2.276000,108.845000,-179.514000,1.248000,137.427000,"
  [245] = "-19.530000,2.126000,108.854000,-179.540000,1.218000,138.567000,"
  [246] = "-19.412000,1.983000,108.864000,-179.565000,1.187000,139.739000,"
  [247] = "-19.297000,1.846000,108.873000,-179.590000,1.156000,140.944000,"
  [248] = "-19.186000,1.714000,108.882000,-179.614000,1.127000,142.182000,"
  [249] = "-19.080000,1.589000,108.891000,-179.637000,1.099000,143.452000,"
  [250] = "-18.979000,1.468000,108.899000,-179.659000,1.072000,144.753000,"
  [251] = "-18.883000,1.345000,108.907000,-179.681000,1.046000,146.050000,"
  [252] = "-18.791000,1.217000,108.915000,-179.701000,1.019000,147.331000,"
  [253] = "-18.703000,1.084000,108.923000,-179.721000,0.992000,148.598000,"
  [254] = "-18.618000,0.946000,108.930000,-179.740000,0.965000,149.852000,"
  [255] = "-18.536000,0.804000,108.938000,-179.758000,0.938000,151.094000,"
  [256] = "-18.457000,0.659000,108.946000,-179.776000,0.909000,152.325000,"
  [257] = "-18.382000,0.509000,108.953000,-179.793000,0.881000,153.546000,"
  [258] = "-18.308000,0.356000,108.961000,-179.809000,0.851000,154.760000,"
  [259] = "-18.238000,0.199000,108.969000,-179.825000,0.821000,155.966000,"
  [260] = "-18.169000,0.039000,108.977000,-179.841000,0.790000,157.167000,"
  [261] = "-18.104000,-0.119000,108.984000,-179.855000,0.758000,158.386000,"
  [262] = "-18.044000,-0.270000,108.992000,-179.869000,0.727000,159.648000,"
  [263] = "-17.988000,-0.416000,108.999000,-179.883000,0.697000,160.955000,"
  [264] = "-17.938000,-0.554000,109.006000,-179.896000,0.667000,162.309000,"
  [265] = "-17.893000,-0.685000,109.013000,-179.909000,0.638000,163.713000,"
  [266] = "-17.854000,-0.808000,109.020000,-179.921000,0.609000,165.171000,"
  [267] = "-17.819000,-0.923000,109.026000,-179.932000,0.581000,166.685000,"
  [268] = "-17.790000,-1.030000,109.032000,-179.943000,0.553000,168.259000,"
  [269] = "-17.766000,-1.128000,109.037000,-179.954000,0.526000,169.896000,"
  [270] = "-17.747000,-1.217000,109.043000,-179.963000,0.499000,171.600000,"
  [271] = "-17.729000,-1.306000,109.048000,-179.973000,0.470000,173.332000,"
  [272] = "-17.710000,-1.401000,109.054000,-179.981000,0.440000,175.061000,"
  [273] = "-17.691000,-1.503000,109.060000,-179.989000,0.407000,176.789000,"
  [274] = "-17.672000,-1.612000,109.066000,-179.995000,0.373000,178.520000,"
  [275] = "-17.656000,-1.728000,109.072000,179.999000,0.338000,-179.741000,"
  [276] = "-17.643000,-1.847000,109.078000,179.995000,0.302000,-177.976000,"
  [277] = "-17.638000,-1.937000,109.083000,179.992000,0.276000,-176.631000,"
  [278] = "-17.638000,-2.029000,109.086000,179.990000,0.251000,-175.263000,"
  [279] = "-17.642000,-2.121000,109.090000,179.988000,0.226000,-173.871000,"
  [280] = "-17.653000,-2.214000,109.093000,179.987000,0.203000,-172.450000,"
  [281] = "-17.668000,-2.309000,109.096000,179.986000,0.181000,-171.012000,"
  [282] = "-17.688000,-2.411000,109.098000,179.985000,0.160000,-169.567000,"
  [283] = "-17.712000,-2.519000,109.100000,179.985000,0.139000,-168.114000,"
  [284] = "-17.741000,-2.634000,109.101000,179.986000,0.120000,-166.653000,"
  [285] = "-17.775000,-2.756000,109.103000,179.987000,0.101000,-165.180000,"
  [286] = "-17.814000,-2.884000,109.103000,179.988000,0.083000,-163.694000,"
  [287] = "-17.860000,-3.020000,109.104000,179.990000,0.066000,-162.192000,"
  [288] = "-17.911000,-3.162000,109.104000,179.992000,0.050000,-160.677000,"
  [289] = "-17.971000,-3.313000,109.103000,179.994000,0.035000,-159.128000,"
  [290] = "-18.037000,-3.468000,109.102000,179.996000,0.022000,-157.586000,"
  [291] = "-18.088000,-3.576000,109.101000,179.997000,0.014000,-156.527000,"
  [292] = "-18.144000,-3.684000,109.099000,179.998000,0.007000,-155.445000,"
  [293] = "-18.206000,-3.795000,109.097000,180.000000,0.002000,-154.337000,"
  [294] = "-18.274000,-3.907000,109.095000,-179.999000,-0.003000,-153.200000,"
  [295] = "-18.349000,-4.020000,109.092000,-179.999000,-0.006000,-152.031000,"
  [296] = "-18.431000,-4.135000,109.089000,-179.998000,-0.008000,-150.826000,"
  [297] = "-18.520000,-4.251000,109.085000,-179.998000,-0.008000,-149.580000,"
  [298] = "-18.619000,-4.369000,109.081000,-179.998000,-0.008000,-148.288000,"
  [299] = "-18.726000,-4.488000,109.076000,-179.998000,-0.006000,-146.943000,"
  [300] = "-18.844000,-4.609000,109.070000,-179.999000,-0.003000,-145.536000,"
  [301] = "-18.974000,-4.731000,109.064000,179.999000,0.002000,-144.053000,"
  [302] = "-19.070000,-4.820000,109.060000,179.998000,0.006000,-142.989000,"
  [303] = "-19.190000,-4.932000,109.054000,179.996000,0.011000,-141.688000,"
  [304] = "-19.313000,-5.049000,109.048000,179.994000,0.016000,-140.393000,"
  [305] = "-19.431000,-5.162000,109.042000,179.992000,0.021000,-139.184000,"
  [306] = "-19.564000,-5.291000,109.035000,179.989000,0.028000,-137.860000,"
  [307] = "-19.689000,-5.411000,109.029000,179.986000,0.034000,-136.673000,"
  [308] = "-19.819000,-5.541000,109.021000,179.983000,0.043000,-135.477000,"
  [309] = "-19.965000,-5.687000,109.013000,179.977000,0.054000,-134.218000,"
  [310] = "-20.089000,-5.808000,109.006000,179.971000,0.066000,-133.222000,"
  [311] = "-20.240000,-5.950000,108.996000,179.963000,0.084000,-132.095000,"
  [312] = "-20.396000,-6.104000,108.986000,179.952000,0.106000,-131.024000,"
  [313] = "-20.534000,-6.268000,108.976000,179.941000,0.127000,-130.130000,"
  [314] = "-20.675000,-6.476000,108.966000,179.929000,0.149000,-129.253000,"
  [315] = "-20.810000,-6.725000,108.955000,179.918000,0.171000,-128.457000,"
  [316] = "-20.918000,-6.986000,108.946000,179.908000,0.188000,-127.832000,"
  [317] = "-21.001000,-7.219000,108.939000,179.901000,0.200000,-127.367000,"
  [318] = "-21.104000,-7.533000,108.930000,179.892000,0.215000,-126.805000,"
  [319] = "-21.199000,-7.860000,108.921000,179.885000,0.228000,-126.291000,"
  [320] = "-21.277000,-8.157000,108.914000,179.879000,0.238000,-125.877000,"
  [321] = "-21.349000,-8.469000,108.908000,179.874000,0.245000,-125.494000,"
  [322] = "-21.427000,-8.830000,108.901000,179.869000,0.252000,-125.075000,"
  [323] = "-21.502000,-9.149000,108.894000,179.864000,0.259000,-124.688000,"
  [324] = "-21.574000,-9.443000,108.888000,179.860000,0.264000,-124.320000,"
  [325] = "-21.658000,-9.768000,108.882000,179.856000,0.270000,-123.897000,"
  [326] = "-21.674000,-9.754000,109.374000,179.852000,0.278000,-123.896000,"
  [327] = "-21.689000,-9.739000,109.866000,179.847000,0.286000,-123.894000,"
  [328] = "-21.702000,-9.727000,110.259000,179.844000,0.293000,-123.892000,"
  [329] = "-21.714000,-9.715000,110.653000,179.841000,0.299000,-123.891000,"
  [330] = "-21.722000,-9.708000,110.888000,179.838000,0.303000,-123.890000,"
  [331] = "-21.733000,-9.698000,111.243000,179.835000,0.309000,-123.889000,"
  [332] = "-21.749000,-9.683000,111.722000,179.831000,0.317000,-123.887000,"
  [333] = "-21.763000,-9.669000,112.170000,179.827000,0.324000,-123.886000,"
  [334] = "-21.776000,-9.658000,112.552000,179.824000,0.330000,-123.884000,"
  [335] = "-21.788000,-9.646000,112.935000,179.821000,0.336000,-123.883000,"
  [336] = "-21.700000,-9.294000,112.942000,179.826000,0.330000,-124.332000,"
  [337] = "-21.618000,-8.955000,112.948000,179.830000,0.324000,-124.748000,"
  [338] = "-21.542000,-8.622000,112.955000,179.836000,0.317000,-125.142000,"
  [339] = "-21.478000,-8.334000,112.960000,179.840000,0.310000,-125.470000,"
  [340] = "-21.404000,-8.005000,112.967000,179.846000,0.301000,-125.849000,"
  [341] = "-21.335000,-7.746000,112.974000,179.852000,0.291000,-126.192000,"
  [342] = "-21.238000,-7.426000,112.982000,179.862000,0.275000,-126.676000,"
  [343] = "-21.133000,-7.122000,112.992000,179.872000,0.258000,-127.210000,"
  [344] = "-21.029000,-6.846000,113.001000,179.882000,0.240000,-127.760000,"
  [345] = "-20.917000,-6.586000,113.010000,179.893000,0.221000,-128.373000,"
  [346] = "-20.776000,-6.336000,113.022000,179.907000,0.197000,-129.170000,"
  [347] = "-20.632000,-6.139000,113.033000,179.920000,0.172000,-130.028000,"
  [348] = "-20.488000,-5.982000,113.043000,179.932000,0.148000,-130.928000,"
  [349] = "-20.307000,-5.830000,113.055000,179.947000,0.120000,-132.114000,"
  [350] = "-20.167000,-5.727000,113.065000,179.957000,0.100000,-133.098000,"
  [351] = "-20.018000,-5.611000,113.074000,179.966000,0.081000,-134.223000,"
  [352] = "-19.869000,-5.488000,113.083000,179.973000,0.066000,-135.426000,"
  [353] = "-19.741000,-5.378000,113.090000,179.978000,0.055000,-136.537000,"
  [354] = "-19.634000,-5.285000,113.096000,179.982000,0.047000,-137.505000,"
  [355] = "-19.504000,-5.171000,113.103000,179.986000,0.038000,-138.734000,"
  [356] = "-19.398000,-5.076000,113.108000,179.988000,0.032000,-139.779000,"
  [357] = "-19.265000,-4.956000,113.115000,179.991000,0.025000,-141.136000,"
  [358] = "-19.138000,-4.839000,113.121000,179.993000,0.019000,-142.492000,"
  [359] = "-19.035000,-4.746000,113.126000,179.995000,0.015000,-143.613000,"
  [360] = "-18.942000,-4.661000,113.130000,179.996000,0.011000,-144.660000,"
  [361] = "-18.814000,-4.540000,113.136000,179.998000,0.007000,-146.145000,"
  [362] = "-18.698000,-4.422000,113.142000,179.999000,0.004000,-147.559000,"
  [363] = "-18.592000,-4.305000,113.146000,179.999000,0.003000,-148.911000,"
  [364] = "-18.496000,-4.189000,113.150000,179.999000,0.003000,-150.210000,"
  [365] = "-18.409000,-4.075000,113.154000,179.999000,0.005000,-151.464000,"
  [366] = "-18.329000,-3.963000,113.157000,179.998000,0.007000,-152.677000,"
  [367] = "-18.256000,-3.853000,113.160000,179.997000,0.011000,-153.855000,"
  [368] = "-18.190000,-3.744000,113.162000,179.996000,0.016000,-155.001000,"
  [369] = "-18.130000,-3.637000,113.164000,179.995000,0.022000,-156.118000,"
  [370] = "-18.076000,-3.532000,113.165000,179.994000,0.029000,-157.210000,"
  [371] = "-18.027000,-3.428000,113.166000,179.993000,0.038000,-158.278000,"
  [372] = "-17.962000,-3.278000,113.167000,179.991000,0.051000,-159.834000,"
  [373] = "-17.904000,-3.133000,113.167000,179.989000,0.066000,-161.391000,"
  [374] = "-17.854000,-2.996000,113.167000,179.988000,0.082000,-162.912000,"
  [375] = "-17.810000,-2.866000,113.167000,179.986000,0.099000,-164.415000,"
  [376] = "-17.772000,-2.744000,113.166000,179.986000,0.117000,-165.902000,"
  [377] = "-17.739000,-2.628000,113.165000,179.985000,0.136000,-167.377000,"
  [378] = "-17.710000,-2.519000,113.163000,179.985000,0.155000,-168.841000,"
  [379] = "-17.687000,-2.416000,113.161000,179.985000,0.175000,-170.297000,"
  [380] = "-17.667000,-2.319000,113.159000,179.986000,0.196000,-171.746000,"
  [381] = "-17.651000,-2.228000,113.156000,179.987000,0.217000,-173.189000,"
  [382] = "-17.641000,-2.140000,113.153000,179.989000,0.240000,-174.615000,"
  [383] = "-17.636000,-2.052000,113.150000,179.991000,0.264000,-176.011000,"
  [384] = "-17.637000,-1.964000,113.146000,179.993000,0.289000,-177.381000,"
  [385] = "-17.644000,-1.877000,113.142000,179.997000,0.315000,-178.727000,"
  [386] = "-17.658000,-1.762000,113.136000,-179.999000,0.351000,179.511000,"
  [387] = "-17.679000,-1.649000,113.129000,-179.992000,0.387000,177.778000,"
  [388] = "-17.703000,-1.541000,113.123000,-179.985000,0.423000,176.057000,"
  [389] = "-17.728000,-1.439000,113.116000,-179.977000,0.458000,174.342000,"
  [390] = "-17.753000,-1.343000,113.110000,-179.968000,0.491000,172.631000,"
  [391] = "-17.776000,-1.253000,113.104000,-179.959000,0.521000,170.920000,"
  [392] = "-17.798000,-1.163000,113.098000,-179.948000,0.549000,169.233000,"
  [393] = "-17.824000,-1.065000,113.092000,-179.937000,0.576000,167.610000,"
  [394] = "-17.854000,-0.958000,113.086000,-179.926000,0.604000,166.047000,"
  [395] = "-17.888000,-0.842000,113.080000,-179.914000,0.631000,164.543000,"
  [396] = "-17.926000,-0.719000,113.074000,-179.902000,0.658000,163.093000,"
  [397] = "-17.970000,-0.588000,113.068000,-179.890000,0.686000,161.695000,"
  [398] = "-18.018000,-0.449000,113.061000,-179.876000,0.714000,160.347000,"
  [399] = "-18.072000,-0.304000,113.054000,-179.863000,0.742000,159.044000,"
  [400] = "-18.131000,-0.153000,113.047000,-179.849000,0.771000,157.785000,"
  [401] = "-18.195000,0.005000,113.039000,-179.834000,0.801000,156.567000,"
  [402] = "-18.263000,0.165000,113.032000,-179.819000,0.831000,155.371000,"
  [403] = "-18.334000,0.321000,113.024000,-179.803000,0.861000,154.168000,"
  [404] = "-18.408000,0.474000,113.016000,-179.786000,0.890000,152.956000,"
  [405] = "-18.485000,0.622000,113.009000,-179.769000,0.918000,151.735000,"
  [406] = "-18.565000,0.767000,113.001000,-179.751000,0.946000,150.504000,"
  [407] = "-18.647000,0.908000,112.994000,-179.733000,0.973000,149.260000,"
  [408] = "-18.734000,1.044000,112.986000,-179.713000,1.000000,148.003000,"
  [409] = "-18.823000,1.175000,112.978000,-179.693000,1.026000,146.732000,"
  [410] = "-18.917000,1.301000,112.970000,-179.673000,1.052000,145.445000,"
  [411] = "-19.014000,1.423000,112.962000,-179.651000,1.078000,144.141000,"
  [412] = "-19.115000,1.541000,112.954000,-179.629000,1.104000,142.831000,"
  [413] = "-19.222000,1.664000,112.945000,-179.605000,1.132000,141.553000,"
  [414] = "-19.306000,1.761000,112.939000,-179.587000,1.153000,140.619000,"
  [415] = "-19.420000,1.896000,112.930000,-179.563000,1.183000,139.405000,"
  [416] = "-19.538000,2.038000,112.920000,-179.537000,1.213000,138.227000,"
  [417] = "-19.659000,2.188000,112.911000,-179.511000,1.243000,137.085000,"
  [418] = "-19.782000,2.346000,112.901000,-179.485000,1.274000,135.980000,"
  [419] = "-19.906000,2.512000,112.892000,-179.459000,1.304000,134.910000,"
  [420] = "-20.030000,2.687000,112.883000,-179.432000,1.333000,133.875000,"
  [421] = "-20.153000,2.871000,112.874000,-179.407000,1.361000,132.874000,"
  [422] = "-20.275000,3.065000,112.865000,-179.381000,1.387000,131.906000,"
  [423] = "-20.394000,3.266000,112.858000,-179.357000,1.410000,130.954000,"
  [424] = "-20.513000,3.471000,112.851000,-179.333000,1.432000,130.012000,"
  [425] = "-20.631000,3.682000,112.844000,-179.309000,1.451000,129.082000,"
  [426] = "-20.750000,3.897000,112.837000,-179.286000,1.469000,128.163000,"
  [427] = "-20.863000,4.107000,112.832000,-179.264000,1.486000,127.301000,"
  [428] = "-20.984000,4.331000,112.826000,-179.241000,1.502000,126.403000,"
  [429] = "-21.108000,4.560000,112.820000,-179.218000,1.518000,125.516000,"
  [430] = "-21.236000,4.793000,112.814000,-179.195000,1.534000,124.640000,"
  [431] = "-21.367000,5.029000,112.808000,-179.171000,1.551000,123.774000,"
  [432] = "-21.503000,5.271000,112.802000,-179.147000,1.569000,122.930000,"
  [433] = "-21.642000,5.523000,112.795000,-179.121000,1.589000,122.126000,"
  [434] = "-21.782000,5.786000,112.789000,-179.096000,1.610000,121.362000,"
  [435] = "-21.922000,6.061000,112.783000,-179.070000,1.632000,120.639000,"
  [436] = "-22.061000,6.347000,112.777000,-179.044000,1.654000,119.962000,"
  [437] = "-22.194000,6.640000,112.771000,-179.020000,1.676000,119.341000,"
  [438] = "-22.306000,6.903000,112.767000,-178.999000,1.694000,118.842000,"
  [439] = "-22.396000,7.129000,112.763000,-178.983000,1.708000,118.450000,"
  [440] = "-22.516000,7.460000,112.759000,-178.961000,1.727000,117.939000,"
  [441] = "-22.614000,7.756000,112.756000,-178.943000,1.742000,117.533000,"
  [442] = "-22.689000,7.999000,112.754000,-178.931000,1.753000,117.223000,"
  [443] = "-22.778000,8.311000,112.753000,-178.916000,1.764000,116.853000,"
  [444] = "-22.846000,8.567000,112.752000,-178.904000,1.773000,116.571000,"
  [445] = "-22.929000,8.894000,112.751000,-178.891000,1.782000,116.235000,"
  [446] = "-22.991000,9.162000,112.750000,-178.882000,1.789000,115.981000,"
  [447] = "-23.067000,9.504000,112.750000,-178.870000,1.797000,115.682000,"
  [448] = "-23.125000,9.783000,112.750000,-178.862000,1.802000,115.457000,"
  [449] = "-23.194000,10.139000,112.751000,-178.852000,1.809000,115.195000,"
  [450] = "-23.248000,10.429000,112.751000,-178.844000,1.815000,115.000000,"
  [451] = "-23.312000,10.798000,112.752000,-178.834000,1.822000,114.775000,"
  [452] = "-23.368000,11.135000,112.753000,-178.826000,1.828000,114.590000,"
  [453] = "-23.424000,11.474000,112.754000,-178.818000,1.835000,114.406000,"
  [454] = "-23.482000,11.814000,112.755000,-178.809000,1.841000,114.219000,"
  [455] = "-23.541000,12.153000,112.756000,-178.801000,1.847000,114.031000,"
  [456] = "-23.601000,12.493000,112.757000,-178.793000,1.853000,113.841000,"
  [457] = "-23.662000,12.834000,112.759000,-178.785000,1.858000,113.649000,"
  [458] = "-23.725000,13.175000,112.760000,-178.777000,1.864000,113.454000,"
  [459] = "-23.789000,13.516000,112.761000,-178.769000,1.869000,113.257000,"
  [460] = "-23.848000,13.820000,112.763000,-178.762000,1.874000,113.081000,"
  [461] = "-23.922000,14.200000,112.764000,-178.753000,1.879000,112.857000,"
  [462] = "-23.983000,14.504000,112.766000,-178.746000,1.883000,112.677000,"
  [463] = "-24.061000,14.885000,112.768000,-178.737000,1.888000,112.448000,"
  [464] = "-24.125000,15.191000,112.769000,-178.730000,1.892000,112.263000,"
  [465] = "-24.207000,15.573000,112.771000,-178.722000,1.896000,112.030000,"
  [466] = "-24.273000,15.879000,112.773000,-178.715000,1.899000,111.841000,"
  [467] = "-24.359000,16.262000,112.775000,-178.707000,1.903000,111.602000,"
  [468] = "-24.428000,16.569000,112.777000,-178.700000,1.906000,111.408000,"
  [469] = "-24.518000,16.953000,112.779000,-178.692000,1.910000,111.164000,"
  [470] = "-24.591000,17.261000,112.781000,-178.685000,1.912000,110.966000,"
  [471] = "-24.684000,17.646000,112.783000,-178.677000,1.915000,110.716000,"
  [472] = "-24.761000,17.954000,112.785000,-178.670000,1.918000,110.513000,"
  [473] = "-24.858000,18.341000,112.787000,-178.662000,1.920000,110.257000,"
  [474] = "-24.938000,18.651000,112.789000,-178.655000,1.922000,110.053000,"
  [475] = "-25.036000,19.042000,112.792000,-178.647000,1.925000,109.803000,"
  [476] = "-25.125000,19.396000,112.794000,-178.640000,1.927000,109.583000,"
  [477] = "-25.213000,19.753000,112.797000,-178.633000,1.929000,109.368000,"
  [478] = "-25.301000,20.113000,112.799000,-178.626000,1.932000,109.158000,"
  [479] = "-25.388000,20.475000,112.802000,-178.619000,1.934000,108.952000,"
  [480] = "-25.475000,20.840000,112.805000,-178.612000,1.937000,108.752000,"
  [481] = "-25.561000,21.208000,112.808000,-178.605000,1.939000,108.556000,"
  [482] = "-25.646000,21.578000,112.811000,-178.599000,1.942000,108.366000,"
  [483] = "-25.731000,21.951000,112.814000,-178.592000,1.945000,108.181000,"
  [484] = "-25.806000,22.284000,112.816000,-178.586000,1.947000,108.017000,"
  [485] = "-25.904000,22.699000,112.820000,-178.578000,1.950000,107.807000,"
  [486] = "-25.985000,23.031000,112.823000,-178.573000,1.951000,107.633000,"
  [487] = "-26.090000,23.446000,112.826000,-178.566000,1.953000,107.408000,"
  [488] = "-26.176000,23.779000,112.829000,-178.561000,1.953000,107.222000,"
  [489] = "-26.285000,24.194000,112.833000,-178.555000,1.952000,106.983000,"
  [490] = "-26.394000,24.598000,112.836000,-178.551000,1.949000,106.744000,"
  [491] = "-26.489000,24.946000,112.839000,-178.548000,1.945000,106.532000,"
  [492] = "-26.600000,25.352000,112.842000,-178.546000,1.939000,106.279000,"
  [493] = "-26.732000,25.679000,112.844000,-178.545000,1.930000,105.976000,"
  [494] = "-26.728000,25.680000,113.344000,-178.545000,1.931000,105.987000,"
  [495] = "-26.724000,25.682000,113.844000,-178.544000,1.931000,105.998000,"
  [496] = "-26.721000,25.683000,114.244000,-178.544000,1.932000,106.007000,"
  [497] = "-26.718000,25.684000,114.644000,-178.544000,1.933000,106.016000,"
  [498] = "-26.716000,25.685000,114.883000,-178.544000,1.933000,106.021000,"
  [499] = "-26.713000,25.686000,115.244000,-178.544000,1.934000,106.029000,"
  [500] = "-26.710000,25.687000,115.719000,-178.543000,1.935000,106.040000,"
  [501] = "-26.706000,25.689000,116.169000,-178.543000,1.935000,106.050000,"
  [502] = "-26.703000,25.690000,116.538000,-178.543000,1.936000,106.058000,"
  [503] = "-26.700000,25.691000,116.907000,-178.542000,1.936000,106.066000,"
  [504] = "-26.604000,25.339000,116.904000,-178.541000,1.947000,106.303000,"
  [505] = "-26.507000,24.922000,116.900000,-178.541000,1.955000,106.534000,"
  [506] = "-26.422000,24.567000,116.897000,-178.543000,1.959000,106.730000,"
  [507] = "-26.321000,24.159000,116.893000,-178.547000,1.962000,106.952000,"
  [508] = "-26.215000,23.739000,116.890000,-178.553000,1.962000,107.177000,"
  [509] = "-26.131000,23.406000,116.887000,-178.558000,1.961000,107.354000,"
  [510] = "-26.026000,22.991000,116.883000,-178.566000,1.958000,107.571000,"
  [511] = "-25.944000,22.659000,116.880000,-178.573000,1.955000,107.742000,"
  [512] = "-25.844000,22.245000,116.877000,-178.581000,1.951000,107.950000,"
  [513] = "-25.766000,21.914000,116.874000,-178.587000,1.948000,108.114000,"
  [514] = "-25.670000,21.501000,116.871000,-178.595000,1.945000,108.322000,"
  [515] = "-25.594000,21.173000,116.868000,-178.601000,1.943000,108.493000,"
  [516] = "-25.498000,20.764000,116.865000,-178.609000,1.940000,108.712000,"
  [517] = "-25.421000,20.440000,116.863000,-178.614000,1.938000,108.891000,"
  [518] = "-25.325000,20.036000,116.859000,-178.622000,1.937000,109.119000,"
  [519] = "-25.249000,19.716000,116.857000,-178.627000,1.935000,109.307000,"
  [520] = "-25.153000,19.318000,116.854000,-178.635000,1.934000,109.545000,"
  [521] = "-25.075000,19.002000,116.852000,-178.640000,1.932000,109.740000,"
  [522] = "-24.979000,18.610000,116.849000,-178.648000,1.931000,109.989000,"
  [523] = "-24.901000,18.298000,116.847000,-178.654000,1.929000,110.192000,"
  [524] = "-24.805000,17.911000,116.845000,-178.662000,1.927000,110.445000,"
  [525] = "-24.729000,17.601000,116.843000,-178.668000,1.925000,110.646000,"
  [526] = "-24.636000,17.216000,116.840000,-178.676000,1.923000,110.894000,"
  [527] = "-24.563000,16.907000,116.838000,-178.683000,1.920000,111.090000,"
  [528] = "-24.474000,16.523000,116.836000,-178.691000,1.916000,111.332000,"
  [529] = "-24.404000,16.216000,116.834000,-178.698000,1.913000,111.524000,"
  [530] = "-24.319000,15.833000,116.832000,-178.706000,1.909000,111.760000,"
  [531] = "-24.251000,15.527000,116.831000,-178.713000,1.905000,111.948000,"
  [532] = "-24.169000,15.145000,116.829000,-178.722000,1.901000,112.179000,"
  [533] = "-24.105000,14.840000,116.827000,-178.729000,1.896000,112.363000,"
  [534] = "-24.026000,14.459000,116.825000,-178.738000,1.891000,112.589000,"
  [535] = "-23.964000,14.155000,116.824000,-178.746000,1.887000,112.768000,"
  [536] = "-23.888000,13.775000,116.822000,-178.755000,1.881000,112.990000,"
  [537] = "-23.829000,13.472000,116.821000,-178.762000,1.876000,113.165000,"
  [538] = "-23.756000,13.093000,116.819000,-178.771000,1.870000,113.382000,"
  [539] = "-23.699000,12.790000,116.818000,-178.779000,1.864000,113.553000,"
  [540] = "-23.630000,12.413000,116.817000,-178.788000,1.858000,113.765000,"
  [541] = "-23.576000,12.111000,116.816000,-178.796000,1.852000,113.933000,"
  [542] = "-23.509000,11.733000,116.815000,-178.805000,1.845000,114.141000,"
  [543] = "-23.458000,11.432000,116.814000,-178.812000,1.839000,114.305000,"
  [544] = "-23.394000,11.056000,116.813000,-178.822000,1.832000,114.508000,"
  [545] = "-23.344000,10.756000,116.812000,-178.829000,1.826000,114.673000,"
  [546] = "-23.280000,10.387000,116.811000,-178.839000,1.819000,114.897000,"
  [547] = "-23.226000,10.096000,116.810000,-178.846000,1.814000,115.089000,"
  [548] = "-23.157000,9.739000,116.810000,-178.857000,1.807000,115.346000,"
  [549] = "-23.100000,9.458000,116.810000,-178.865000,1.801000,115.564000,"
  [550] = "-23.025000,9.114000,116.810000,-178.876000,1.793000,115.854000,"
  [551] = "-22.963000,8.844000,116.810000,-178.886000,1.786000,116.098000,"
  [552] = "-22.882000,8.513000,116.811000,-178.899000,1.776000,116.419000,"
  [553] = "-22.814000,8.255000,116.812000,-178.910000,1.767000,116.689000,"
  [554] = "-22.725000,7.939000,116.814000,-178.925000,1.755000,117.041000,"
  [555] = "-22.651000,7.692000,116.816000,-178.938000,1.744000,117.335000,"
  [556] = "-22.553000,7.392000,116.819000,-178.956000,1.728000,117.720000,"
  [557] = "-22.432000,7.057000,116.823000,-178.978000,1.707000,118.214000,"
  [558] = "-22.341000,6.829000,116.826000,-178.995000,1.692000,118.596000,"
  [559] = "-22.228000,6.565000,116.831000,-179.016000,1.674000,119.085000,"
  [560] = "-22.093000,6.271000,116.837000,-179.041000,1.651000,119.699000,"
  [561] = "-21.995000,6.070000,116.841000,-179.059000,1.636000,120.165000,"
  [562] = "-21.877000,5.837000,116.846000,-179.081000,1.617000,120.755000,"
  [563] = "-21.738000,5.577000,116.852000,-179.106000,1.596000,121.483000,"
  [564] = "-21.597000,5.323000,116.859000,-179.131000,1.576000,122.272000,"
  [565] = "-21.458000,5.079000,116.865000,-179.156000,1.557000,123.108000,"
  [566] = "-21.323000,4.843000,116.871000,-179.180000,1.541000,123.977000,"
  [567] = "-21.193000,4.610000,116.877000,-179.204000,1.525000,124.853000,"
  [568] = "-21.066000,4.380000,116.883000,-179.227000,1.509000,125.736000,"
  [569] = "-20.943000,4.153000,116.889000,-179.250000,1.492000,126.626000,"
  [570] = "-20.822000,3.929000,116.895000,-179.273000,1.476000,127.524000,"
  [571] = "-20.702000,3.710000,116.901000,-179.296000,1.458000,128.429000,"
  [572] = "-20.583000,3.494000,116.908000,-179.319000,1.438000,129.342000,"
  [573] = "-20.469000,3.294000,116.914000,-179.342000,1.418000,130.216000,"
  [574] = "-20.348000,3.088000,116.922000,-179.366000,1.395000,131.144000,"
  [575] = "-20.226000,2.886000,116.930000,-179.392000,1.369000,132.081000,"
  [576] = "-20.102000,2.694000,116.939000,-179.418000,1.341000,133.050000,"
  [577] = "-19.976000,2.513000,116.948000,-179.444000,1.312000,134.057000,"
  [578] = "-19.851000,2.342000,116.957000,-179.470000,1.283000,135.104000,"
  [579] = "-19.727000,2.180000,116.967000,-179.496000,1.252000,136.189000,"
  [580] = "-19.605000,2.027000,116.976000,-179.522000,1.222000,137.314000,"
  [581] = "-19.485000,1.882000,116.986000,-179.548000,1.192000,138.478000,"
  [582] = "-19.397000,1.779000,116.993000,-179.567000,1.170000,139.378000,"
  [583] = "-19.311000,1.680000,116.999000,-179.585000,1.149000,140.300000,"
  [584] = "-19.201000,1.555000,117.008000,-179.609000,1.121000,141.564000,"
  [585] = "-19.096000,1.436000,117.016000,-179.632000,1.095000,142.867000,"
  [586] = "-18.996000,1.319000,117.024000,-179.654000,1.070000,144.186000,"
  [587] = "-18.900000,1.197000,117.032000,-179.676000,1.044000,145.487000,"
  [588] = "-18.806000,1.070000,117.040000,-179.696000,1.018000,146.770000,"
  [589] = "-18.717000,0.938000,117.048000,-179.716000,0.992000,148.037000,"
  [590] = "-18.631000,0.802000,117.056000,-179.735000,0.965000,149.290000,"
  [591] = "-18.548000,0.660000,117.063000,-179.753000,0.937000,150.529000,"
  [592] = "-18.468000,0.515000,117.071000,-179.771000,0.910000,151.756000,"
  [593] = "-18.391000,0.365000,117.078000,-179.788000,0.881000,152.972000,"
  [594] = "-18.318000,0.211000,117.086000,-179.805000,0.853000,154.178000,"
  [595] = "-18.247000,0.054000,117.094000,-179.820000,0.824000,155.376000,"
  [596] = "-18.181000,-0.105000,117.101000,-179.835000,0.794000,156.577000,"
  [597] = "-18.120000,-0.259000,117.108000,-179.850000,0.766000,157.814000,"
  [598] = "-18.065000,-0.407000,117.115000,-179.864000,0.739000,159.092000,"
  [599] = "-18.015000,-0.548000,117.121000,-179.877000,0.712000,160.413000,"
  [600] = "-17.970000,-0.683000,117.128000,-179.890000,0.685000,161.779000,"
  [601] = "-17.929000,-0.811000,117.134000,-179.903000,0.659000,163.193000,"
  [602] = "-17.893000,-0.932000,117.140000,-179.915000,0.633000,164.657000,"
  [603] = "-17.860000,-1.044000,117.146000,-179.927000,0.606000,166.175000,"
  [604] = "-17.831000,-1.149000,117.152000,-179.938000,0.579000,167.750000,"
  [605] = "-17.804000,-1.245000,117.158000,-179.949000,0.550000,169.383000,"
  [606] = "-17.778000,-1.336000,117.164000,-179.959000,0.520000,171.064000,"
  [607] = "-17.748000,-1.431000,117.170000,-179.969000,0.487000,172.752000,"
  [608] = "-17.718000,-1.530000,117.177000,-179.978000,0.452000,174.448000,"
  [609] = "-17.689000,-1.634000,117.184000,-179.986000,0.415000,176.154000,"
  [610] = "-17.663000,-1.742000,117.191000,-179.993000,0.378000,177.876000,"
  [611] = "-17.643000,-1.853000,117.198000,-179.999000,0.341000,179.622000,"
  [612] = "-17.631000,-1.964000,117.204000,179.996000,0.306000,-178.596000,"
  [613] = "-17.627000,-2.048000,117.208000,179.993000,0.281000,-177.232000,"
  [614] = "-17.630000,-2.132000,117.211000,179.991000,0.257000,-175.841000,"
  [615] = "-17.639000,-2.215000,117.214000,179.989000,0.235000,-174.421000,"
  [616] = "-17.653000,-2.300000,117.217000,179.987000,0.214000,-172.976000,"
  [617] = "-17.671000,-2.390000,117.219000,179.986000,0.194000,-171.526000,"
  [618] = "-17.693000,-2.486000,117.221000,179.985000,0.174000,-170.070000,"
  [619] = "-17.720000,-2.588000,117.223000,179.985000,0.154000,-168.606000,"
  [620] = "-17.750000,-2.696000,117.225000,179.985000,0.136000,-167.134000,"
  [621] = "-17.785000,-2.811000,117.226000,179.985000,0.118000,-165.650000,"
  [622] = "-17.826000,-2.933000,117.226000,179.986000,0.101000,-164.153000,"
  [623] = "-17.872000,-3.061000,117.227000,179.987000,0.084000,-162.639000,"
  [624] = "-17.925000,-3.196000,117.226000,179.989000,0.069000,-161.112000,"
  [625] = "-17.985000,-3.339000,117.226000,179.990000,0.054000,-159.547000,"
  [626] = "-18.052000,-3.484000,117.225000,179.992000,0.042000,-157.989000,"
  [627] = "-18.103000,-3.584000,117.223000,179.993000,0.034000,-156.914000,"
  [628] = "-18.160000,-3.686000,117.222000,179.994000,0.028000,-155.815000,"
  [629] = "-18.222000,-3.789000,117.220000,179.995000,0.022000,-154.691000,"
  [630] = "-18.290000,-3.893000,117.218000,179.996000,0.017000,-153.539000,"
  [631] = "-18.365000,-3.999000,117.215000,179.997000,0.014000,-152.355000,"
  [632] = "-18.446000,-4.107000,117.212000,179.997000,0.011000,-151.136000,"
  [633] = "-18.535000,-4.216000,117.208000,179.997000,0.010000,-149.877000,"
  [634] = "-18.633000,-4.327000,117.204000,179.997000,0.010000,-148.573000,"
  [635] = "-18.740000,-4.439000,117.199000,179.996000,0.012000,-147.217000,"
  [636] = "-18.858000,-4.553000,117.194000,179.995000,0.015000,-145.799000,"
  [637] = "-18.988000,-4.669000,117.188000,179.994000,0.020000,-144.312000,"
  [638] = "-19.084000,-4.754000,117.183000,179.992000,0.024000,-143.254000,"
  [639] = "-19.205000,-4.860000,117.177000,179.990000,0.030000,-141.952000,"
  [640] = "-19.331000,-4.968000,117.171000,179.987000,0.037000,-140.654000,"
  [641] = "-19.454000,-5.071000,117.165000,179.983000,0.045000,-139.438000,"
  [642] = "-19.597000,-5.186000,117.157000,179.979000,0.055000,-138.098000,"
  [643] = "-19.731000,-5.289000,117.150000,179.974000,0.067000,-136.902000,"
  [644] = "-19.878000,-5.397000,117.141000,179.967000,0.082000,-135.669000,"
  [645] = "-20.046000,-5.511000,117.131000,179.957000,0.102000,-134.357000,"
  [646] = "-20.191000,-5.602000,117.122000,179.947000,0.122000,-133.296000,"
  [647] = "-20.367000,-5.705000,117.110000,179.934000,0.149000,-132.102000,"
  [648] = "-20.519000,-5.814000,117.100000,179.921000,0.174000,-131.127000,"
  [649] = "-20.699000,-5.986000,117.087000,179.904000,0.205000,-130.024000,"
  [650] = "-20.858000,-6.190000,117.075000,179.889000,0.233000,-129.097000,"
  [651] = "-21.001000,-6.437000,117.063000,179.875000,0.259000,-128.303000,"
  [652] = "-21.119000,-6.698000,117.053000,179.862000,0.280000,-127.683000,"
  [653] = "-21.234000,-6.983000,117.043000,179.850000,0.301000,-127.107000,"
  [654] = "-21.330000,-7.253000,117.034000,179.840000,0.319000,-126.638000,"
  [655] = "-21.434000,-7.593000,117.025000,179.829000,0.337000,-126.141000,"
  [656] = "-21.511000,-7.900000,117.018000,179.821000,0.349000,-125.768000,"
  [657] = "-21.578000,-8.217000,117.011000,179.816000,0.357000,-125.430000,"
  [658] = "-21.658000,-8.588000,117.004000,179.810000,0.366000,-125.020000,"
  [659] = "-21.732000,-8.918000,116.998000,179.805000,0.372000,-124.641000,"
  [660] = "-21.801000,-9.216000,116.992000,179.801000,0.377000,-124.284000,"
  [661] = "-21.876000,-9.530000,116.987000,179.797000,0.381000,-123.897000,"
  [662] = "-21.882000,-9.521000,117.484000,179.795000,0.384000,-123.896000,"
  [663] = "-21.888000,-9.513000,117.981000,179.794000,0.387000,-123.895000,"
  [664] = "-21.893000,-9.506000,118.379000,179.792000,0.389000,-123.894000,"
  [665] = "-21.898000,-9.499000,118.777000,179.791000,0.392000,-123.893000,"
  [666] = "-21.901000,-9.495000,119.014000,179.790000,0.393000,-123.892000,"
  [667] = "-21.906000,-9.489000,119.373000,179.789000,0.396000,-123.892000,"
  [668] = "-21.912000,-9.481000,119.848000,179.788000,0.398000,-123.891000,"
  [669] = "-21.918000,-9.473000,120.297000,179.786000,0.401000,-123.890000,"
  [670] = "-21.923000,-9.467000,120.668000,179.785000,0.403000,-123.889000,"
  [671] = "-21.928000,-9.460000,121.039000,179.784000,0.406000,-123.888000,"
  [672] = "-21.845000,-9.093000,121.045000,179.788000,0.402000,-124.325000,"
